DATA_BLOCK "n0008-icg12-el001-k30001_SN51_3"   // DB1076, F_DB
VERSION : 0.1
// stored: AutoNumber true, DBAccessibleFromOPCUA true, DBAccessibleFromWebserver true, InstanceOfName 00_Push-Button_Input, InstanceOfType FB
"00_Push-Button_Input"
   // VAR_INPUT
   //    IN_1 : Bool;
   //    IN_2 : Bool;
   //    IN_3 : Bool;
   //    IN_4 : Bool;
   //    ON_Tristate : Bool;
   //    ON_Lamp : Bool;
   //    Reset : Bool;
   //    REAC_DELAY { ExternalWritable := 'False'} : Time;
   //    Bypass_ET200 : Bool;
   // END_VAR
   // VAR_OUTPUT
   //    OUT_1 : Bool;
   //    OUT_2 : Bool;
   //    OUT_3 : Bool;
   //    OUT_4 : Bool;
   //    Diag_1 : Bool;
   //    Diag_2 : Bool;
   //    Diag_3 : Bool;
   //    Diag_4 : Bool;
   //    Lamp_1 : Bool;
   //    Lamp_2 : Bool;
   //    Lamp_3 : Bool;
   //    Lamp_4 : Bool;
   // END_VAR
   // VAR
   //    ESTOP_1 { S7_SetPoint := 'True'} : ESTOP1;
   //    ESTOP_2 { S7_SetPoint := 'True'} : ESTOP1;
   //    ESTOP_3 { S7_SetPoint := 'True'} : ESTOP1;
   //    ESTOP_4 { S7_SetPoint := 'True'} : ESTOP1;
   //    TON_1 { ExternalWritable := 'False'} : TON;
   //    TON_2 { ExternalWritable := 'False'} : TON;
   //    TON_3 { ExternalWritable := 'False'} : TON;
   //    TON_4 { ExternalWritable := 'False'} : TON;
   // END_VAR
BEGIN
END_DATA_BLOCK

DATA_BLOCK "n0008-icg12-el001-k30001_SN51_4"   // DB1077, F_DB
VERSION : 0.1
// stored: AutoNumber true, DBAccessibleFromOPCUA true, DBAccessibleFromWebserver true, InstanceOfName 00_Push-Button_Input, InstanceOfType FB
"00_Push-Button_Input"
   // VAR_INPUT
   //    IN_1 : Bool;
   //    IN_2 : Bool;
   //    IN_3 : Bool;
   //    IN_4 : Bool;
   //    ON_Tristate : Bool;
   //    ON_Lamp : Bool;
   //    Reset : Bool;
   //    REAC_DELAY { ExternalWritable := 'False'} : Time;
   //    Bypass_ET200 : Bool;
   // END_VAR
   // VAR_OUTPUT
   //    OUT_1 : Bool;
   //    OUT_2 : Bool;
   //    OUT_3 : Bool;
   //    OUT_4 : Bool;
   //    Diag_1 : Bool;
   //    Diag_2 : Bool;
   //    Diag_3 : Bool;
   //    Diag_4 : Bool;
   //    Lamp_1 : Bool;
   //    Lamp_2 : Bool;
   //    Lamp_3 : Bool;
   //    Lamp_4 : Bool;
   // END_VAR
   // VAR
   //    ESTOP_1 { S7_SetPoint := 'True'} : ESTOP1;
   //    ESTOP_2 { S7_SetPoint := 'True'} : ESTOP1;
   //    ESTOP_3 { S7_SetPoint := 'True'} : ESTOP1;
   //    ESTOP_4 { S7_SetPoint := 'True'} : ESTOP1;
   //    TON_1 { ExternalWritable := 'False'} : TON;
   //    TON_2 { ExternalWritable := 'False'} : TON;
   //    TON_3 { ExternalWritable := 'False'} : TON;
   //    TON_4 { ExternalWritable := 'False'} : TON;
   // END_VAR
BEGIN
END_DATA_BLOCK

DATA_BLOCK "n0026-uc915-xn10_SN51_1"   // DB1078, F_DB
VERSION : 0.1
// stored: AutoNumber true, DBAccessibleFromOPCUA true, DBAccessibleFromWebserver true, InstanceOfName 00_Push-Button_Input, InstanceOfType FB
"00_Push-Button_Input"
   // VAR_INPUT
   //    IN_1 : Bool;
   //    IN_2 : Bool;
   //    IN_3 : Bool;
   //    IN_4 : Bool;
   //    ON_Tristate : Bool;
   //    ON_Lamp : Bool;
   //    Reset : Bool;
   //    REAC_DELAY { ExternalWritable := 'False'} : Time;
   //    Bypass_ET200 : Bool;
   // END_VAR
   // VAR_OUTPUT
   //    OUT_1 : Bool;
   //    OUT_2 : Bool;
   //    OUT_3 : Bool;
   //    OUT_4 : Bool;
   //    Diag_1 : Bool;
   //    Diag_2 : Bool;
   //    Diag_3 : Bool;
   //    Diag_4 : Bool;
   //    Lamp_1 : Bool;
   //    Lamp_2 : Bool;
   //    Lamp_3 : Bool;
   //    Lamp_4 : Bool;
   // END_VAR
   // VAR
   //    ESTOP_1 { S7_SetPoint := 'True'} : ESTOP1;
   //    ESTOP_2 { S7_SetPoint := 'True'} : ESTOP1;
   //    ESTOP_3 { S7_SetPoint := 'True'} : ESTOP1;
   //    ESTOP_4 { S7_SetPoint := 'True'} : ESTOP1;
   //    TON_1 { ExternalWritable := 'False'} : TON;
   //    TON_2 { ExternalWritable := 'False'} : TON;
   //    TON_3 { ExternalWritable := 'False'} : TON;
   //    TON_4 { ExternalWritable := 'False'} : TON;
   // END_VAR
BEGIN
END_DATA_BLOCK

DATA_BLOCK "n0026-uc915-xn10_SN51_2"   // DB1079, F_DB
VERSION : 0.1
// stored: AutoNumber true, DBAccessibleFromOPCUA true, DBAccessibleFromWebserver true, InstanceOfName 00_Push-Button_Input, InstanceOfType FB
"00_Push-Button_Input"
   // VAR_INPUT
   //    IN_1 : Bool;
   //    IN_2 : Bool;
   //    IN_3 : Bool;
   //    IN_4 : Bool;
   //    ON_Tristate : Bool;
   //    ON_Lamp : Bool;
   //    Reset : Bool;
   //    REAC_DELAY { ExternalWritable := 'False'} : Time;
   //    Bypass_ET200 : Bool;
   // END_VAR
   // VAR_OUTPUT
   //    OUT_1 : Bool;
   //    OUT_2 : Bool;
   //    OUT_3 : Bool;
   //    OUT_4 : Bool;
   //    Diag_1 : Bool;
   //    Diag_2 : Bool;
   //    Diag_3 : Bool;
   //    Diag_4 : Bool;
   //    Lamp_1 : Bool;
   //    Lamp_2 : Bool;
   //    Lamp_3 : Bool;
   //    Lamp_4 : Bool;
   // END_VAR
   // VAR
   //    ESTOP_1 { S7_SetPoint := 'True'} : ESTOP1;
   //    ESTOP_2 { S7_SetPoint := 'True'} : ESTOP1;
   //    ESTOP_3 { S7_SetPoint := 'True'} : ESTOP1;
   //    ESTOP_4 { S7_SetPoint := 'True'} : ESTOP1;
   //    TON_1 { ExternalWritable := 'False'} : TON;
   //    TON_2 { ExternalWritable := 'False'} : TON;
   //    TON_3 { ExternalWritable := 'False'} : TON;
   //    TON_4 { ExternalWritable := 'False'} : TON;
   // END_VAR
BEGIN
END_DATA_BLOCK

DATA_BLOCK "n0027-uc915-xn11_SN51_1"   // DB1080, F_DB
VERSION : 0.1
// stored: AutoNumber true, DBAccessibleFromOPCUA true, DBAccessibleFromWebserver true, InstanceOfName 00_Push-Button_Input, InstanceOfType FB
"00_Push-Button_Input"
   // VAR_INPUT
   //    IN_1 : Bool;
   //    IN_2 : Bool;
   //    IN_3 : Bool;
   //    IN_4 : Bool;
   //    ON_Tristate : Bool;
   //    ON_Lamp : Bool;
   //    Reset : Bool;
   //    REAC_DELAY { ExternalWritable := 'False'} : Time;
   //    Bypass_ET200 : Bool;
   // END_VAR
   // VAR_OUTPUT
   //    OUT_1 : Bool;
   //    OUT_2 : Bool;
   //    OUT_3 : Bool;
   //    OUT_4 : Bool;
   //    Diag_1 : Bool;
   //    Diag_2 : Bool;
   //    Diag_3 : Bool;
   //    Diag_4 : Bool;
   //    Lamp_1 : Bool;
   //    Lamp_2 : Bool;
   //    Lamp_3 : Bool;
   //    Lamp_4 : Bool;
   // END_VAR
   // VAR
   //    ESTOP_1 { S7_SetPoint := 'True'} : ESTOP1;
   //    ESTOP_2 { S7_SetPoint := 'True'} : ESTOP1;
   //    ESTOP_3 { S7_SetPoint := 'True'} : ESTOP1;
   //    ESTOP_4 { S7_SetPoint := 'True'} : ESTOP1;
   //    TON_1 { ExternalWritable := 'False'} : TON;
   //    TON_2 { ExternalWritable := 'False'} : TON;
   //    TON_3 { ExternalWritable := 'False'} : TON;
   //    TON_4 { ExternalWritable := 'False'} : TON;
   // END_VAR
BEGIN
END_DATA_BLOCK

DATA_BLOCK "n0029-ct2-el001-k30001_SN51_1"   // DB1081, F_DB
VERSION : 0.1
// stored: AutoNumber true, DBAccessibleFromOPCUA true, DBAccessibleFromWebserver true, InstanceOfName 00_Push-Button_Input, InstanceOfType FB
"00_Push-Button_Input"
   // VAR_INPUT
   //    IN_1 : Bool;
   //    IN_2 : Bool;
   //    IN_3 : Bool;
   //    IN_4 : Bool;
   //    ON_Tristate : Bool;
   //    ON_Lamp : Bool;
   //    Reset : Bool;
   //    REAC_DELAY { ExternalWritable := 'False'} : Time;
   //    Bypass_ET200 : Bool;
   // END_VAR
   // VAR_OUTPUT
   //    OUT_1 : Bool;
   //    OUT_2 : Bool;
   //    OUT_3 : Bool;
   //    OUT_4 : Bool;
   //    Diag_1 : Bool;
   //    Diag_2 : Bool;
   //    Diag_3 : Bool;
   //    Diag_4 : Bool;
   //    Lamp_1 : Bool;
   //    Lamp_2 : Bool;
   //    Lamp_3 : Bool;
   //    Lamp_4 : Bool;
   // END_VAR
   // VAR
   //    ESTOP_1 { S7_SetPoint := 'True'} : ESTOP1;
   //    ESTOP_2 { S7_SetPoint := 'True'} : ESTOP1;
   //    ESTOP_3 { S7_SetPoint := 'True'} : ESTOP1;
   //    ESTOP_4 { S7_SetPoint := 'True'} : ESTOP1;
   //    TON_1 { ExternalWritable := 'False'} : TON;
   //    TON_2 { ExternalWritable := 'False'} : TON;
   //    TON_3 { ExternalWritable := 'False'} : TON;
   //    TON_4 { ExternalWritable := 'False'} : TON;
   // END_VAR
BEGIN
END_DATA_BLOCK

DATA_BLOCK "n0029-ct2-el001-k30001_SN51_2"   // DB1082, F_DB
VERSION : 0.1
// stored: AutoNumber true, DBAccessibleFromOPCUA true, DBAccessibleFromWebserver true, InstanceOfName 00_Push-Button_Input, InstanceOfType FB
"00_Push-Button_Input"
   // VAR_INPUT
   //    IN_1 : Bool;
   //    IN_2 : Bool;
   //    IN_3 : Bool;
   //    IN_4 : Bool;
   //    ON_Tristate : Bool;
   //    ON_Lamp : Bool;
   //    Reset : Bool;
   //    REAC_DELAY { ExternalWritable := 'False'} : Time;
   //    Bypass_ET200 : Bool;
   // END_VAR
   // VAR_OUTPUT
   //    OUT_1 : Bool;
   //    OUT_2 : Bool;
   //    OUT_3 : Bool;
   //    OUT_4 : Bool;
   //    Diag_1 : Bool;
   //    Diag_2 : Bool;
   //    Diag_3 : Bool;
   //    Diag_4 : Bool;
   //    Lamp_1 : Bool;
   //    Lamp_2 : Bool;
   //    Lamp_3 : Bool;
   //    Lamp_4 : Bool;
   // END_VAR
   // VAR
   //    ESTOP_1 { S7_SetPoint := 'True'} : ESTOP1;
   //    ESTOP_2 { S7_SetPoint := 'True'} : ESTOP1;
   //    ESTOP_3 { S7_SetPoint := 'True'} : ESTOP1;
   //    ESTOP_4 { S7_SetPoint := 'True'} : ESTOP1;
   //    TON_1 { ExternalWritable := 'False'} : TON;
   //    TON_2 { ExternalWritable := 'False'} : TON;
   //    TON_3 { ExternalWritable := 'False'} : TON;
   //    TON_4 { ExternalWritable := 'False'} : TON;
   // END_VAR
BEGIN
END_DATA_BLOCK

DATA_BLOCK "n0029-ct2-el001-k30001_SN51_3"   // DB1083, F_DB
VERSION : 0.1
// stored: AutoNumber true, DBAccessibleFromOPCUA true, DBAccessibleFromWebserver true, InstanceOfName 00_Push-Button_Input, InstanceOfType FB
"00_Push-Button_Input"
   // VAR_INPUT
   //    IN_1 : Bool;
   //    IN_2 : Bool;
   //    IN_3 : Bool;
   //    IN_4 : Bool;
   //    ON_Tristate : Bool;
   //    ON_Lamp : Bool;
   //    Reset : Bool;
   //    REAC_DELAY { ExternalWritable := 'False'} : Time;
   //    Bypass_ET200 : Bool;
   // END_VAR
   // VAR_OUTPUT
   //    OUT_1 : Bool;
   //    OUT_2 : Bool;
   //    OUT_3 : Bool;
   //    OUT_4 : Bool;
   //    Diag_1 : Bool;
   //    Diag_2 : Bool;
   //    Diag_3 : Bool;
   //    Diag_4 : Bool;
   //    Lamp_1 : Bool;
   //    Lamp_2 : Bool;
   //    Lamp_3 : Bool;
   //    Lamp_4 : Bool;
   // END_VAR
   // VAR
   //    ESTOP_1 { S7_SetPoint := 'True'} : ESTOP1;
   //    ESTOP_2 { S7_SetPoint := 'True'} : ESTOP1;
   //    ESTOP_3 { S7_SetPoint := 'True'} : ESTOP1;
   //    ESTOP_4 { S7_SetPoint := 'True'} : ESTOP1;
   //    TON_1 { ExternalWritable := 'False'} : TON;
   //    TON_2 { ExternalWritable := 'False'} : TON;
   //    TON_3 { ExternalWritable := 'False'} : TON;
   //    TON_4 { ExternalWritable := 'False'} : TON;
   // END_VAR
BEGIN
END_DATA_BLOCK

DATA_BLOCK "n0029-ct2-el001-k30001_SN51_4"   // DB1084, F_DB
VERSION : 0.1
// stored: AutoNumber true, DBAccessibleFromOPCUA true, DBAccessibleFromWebserver true, InstanceOfName 00_Push-Button_Input, InstanceOfType FB
"00_Push-Button_Input"
   // VAR_INPUT
   //    IN_1 : Bool;
   //    IN_2 : Bool;
   //    IN_3 : Bool;
   //    IN_4 : Bool;
   //    ON_Tristate : Bool;
   //    ON_Lamp : Bool;
   //    Reset : Bool;
   //    REAC_DELAY { ExternalWritable := 'False'} : Time;
   //    Bypass_ET200 : Bool;
   // END_VAR
   // VAR_OUTPUT
   //    OUT_1 : Bool;
   //    OUT_2 : Bool;
   //    OUT_3 : Bool;
   //    OUT_4 : Bool;
   //    Diag_1 : Bool;
   //    Diag_2 : Bool;
   //    Diag_3 : Bool;
   //    Diag_4 : Bool;
   //    Lamp_1 : Bool;
   //    Lamp_2 : Bool;
   //    Lamp_3 : Bool;
   //    Lamp_4 : Bool;
   // END_VAR
   // VAR
   //    ESTOP_1 { S7_SetPoint := 'True'} : ESTOP1;
   //    ESTOP_2 { S7_SetPoint := 'True'} : ESTOP1;
   //    ESTOP_3 { S7_SetPoint := 'True'} : ESTOP1;
   //    ESTOP_4 { S7_SetPoint := 'True'} : ESTOP1;
   //    TON_1 { ExternalWritable := 'False'} : TON;
   //    TON_2 { ExternalWritable := 'False'} : TON;
   //    TON_3 { ExternalWritable := 'False'} : TON;
   //    TON_4 { ExternalWritable := 'False'} : TON;
   // END_VAR
BEGIN
END_DATA_BLOCK

DATA_BLOCK "n0029-ct2-el001-k30001_SN51_5"   // DB1085, F_DB
VERSION : 0.1
// stored: AutoNumber true, DBAccessibleFromOPCUA true, DBAccessibleFromWebserver true, InstanceOfName 00_Push-Button_Input, InstanceOfType FB
"00_Push-Button_Input"
   // VAR_INPUT
   //    IN_1 : Bool;
   //    IN_2 : Bool;
   //    IN_3 : Bool;
   //    IN_4 : Bool;
   //    ON_Tristate : Bool;
   //    ON_Lamp : Bool;
   //    Reset : Bool;
   //    REAC_DELAY { ExternalWritable := 'False'} : Time;
   //    Bypass_ET200 : Bool;
   // END_VAR
   // VAR_OUTPUT
   //    OUT_1 : Bool;
   //    OUT_2 : Bool;
   //    OUT_3 : Bool;
   //    OUT_4 : Bool;
   //    Diag_1 : Bool;
   //    Diag_2 : Bool;
   //    Diag_3 : Bool;
   //    Diag_4 : Bool;
   //    Lamp_1 : Bool;
   //    Lamp_2 : Bool;
   //    Lamp_3 : Bool;
   //    Lamp_4 : Bool;
   // END_VAR
   // VAR
   //    ESTOP_1 { S7_SetPoint := 'True'} : ESTOP1;
   //    ESTOP_2 { S7_SetPoint := 'True'} : ESTOP1;
   //    ESTOP_3 { S7_SetPoint := 'True'} : ESTOP1;
   //    ESTOP_4 { S7_SetPoint := 'True'} : ESTOP1;
   //    TON_1 { ExternalWritable := 'False'} : TON;
   //    TON_2 { ExternalWritable := 'False'} : TON;
   //    TON_3 { ExternalWritable := 'False'} : TON;
   //    TON_4 { ExternalWritable := 'False'} : TON;
   // END_VAR
BEGIN
END_DATA_BLOCK

DATA_BLOCK "n0033-uc26-el001-k30001_SN51_1"   // DB1086, F_DB
VERSION : 0.1
// stored: AutoNumber true, DBAccessibleFromOPCUA true, DBAccessibleFromWebserver true, InstanceOfName 00_Push-Button_Input, InstanceOfType FB
"00_Push-Button_Input"
   // VAR_INPUT
   //    IN_1 : Bool;
   //    IN_2 : Bool;
   //    IN_3 : Bool;
   //    IN_4 : Bool;
   //    ON_Tristate : Bool;
   //    ON_Lamp : Bool;
   //    Reset : Bool;
   //    REAC_DELAY { ExternalWritable := 'False'} : Time;
   //    Bypass_ET200 : Bool;
   // END_VAR
   // VAR_OUTPUT
   //    OUT_1 : Bool;
   //    OUT_2 : Bool;
   //    OUT_3 : Bool;
   //    OUT_4 : Bool;
   //    Diag_1 : Bool;
   //    Diag_2 : Bool;
   //    Diag_3 : Bool;
   //    Diag_4 : Bool;
   //    Lamp_1 : Bool;
   //    Lamp_2 : Bool;
   //    Lamp_3 : Bool;
   //    Lamp_4 : Bool;
   // END_VAR
   // VAR
   //    ESTOP_1 { S7_SetPoint := 'True'} : ESTOP1;
   //    ESTOP_2 { S7_SetPoint := 'True'} : ESTOP1;
   //    ESTOP_3 { S7_SetPoint := 'True'} : ESTOP1;
   //    ESTOP_4 { S7_SetPoint := 'True'} : ESTOP1;
   //    TON_1 { ExternalWritable := 'False'} : TON;
   //    TON_2 { ExternalWritable := 'False'} : TON;
   //    TON_3 { ExternalWritable := 'False'} : TON;
   //    TON_4 { ExternalWritable := 'False'} : TON;
   // END_VAR
BEGIN
END_DATA_BLOCK

DATA_BLOCK "n0033-uc26-el001-k30001_SN51_2"   // DB1087, F_DB
VERSION : 0.1
// stored: AutoNumber true, DBAccessibleFromOPCUA true, DBAccessibleFromWebserver true, InstanceOfName 00_Push-Button_Input, InstanceOfType FB
"00_Push-Button_Input"
   // VAR_INPUT
   //    IN_1 : Bool;
   //    IN_2 : Bool;
   //    IN_3 : Bool;
   //    IN_4 : Bool;
   //    ON_Tristate : Bool;
   //    ON_Lamp : Bool;
   //    Reset : Bool;
   //    REAC_DELAY { ExternalWritable := 'False'} : Time;
   //    Bypass_ET200 : Bool;
   // END_VAR
   // VAR_OUTPUT
   //    OUT_1 : Bool;
   //    OUT_2 : Bool;
   //    OUT_3 : Bool;
   //    OUT_4 : Bool;
   //    Diag_1 : Bool;
   //    Diag_2 : Bool;
   //    Diag_3 : Bool;
   //    Diag_4 : Bool;
   //    Lamp_1 : Bool;
   //    Lamp_2 : Bool;
   //    Lamp_3 : Bool;
   //    Lamp_4 : Bool;
   // END_VAR
   // VAR
   //    ESTOP_1 { S7_SetPoint := 'True'} : ESTOP1;
   //    ESTOP_2 { S7_SetPoint := 'True'} : ESTOP1;
   //    ESTOP_3 { S7_SetPoint := 'True'} : ESTOP1;
   //    ESTOP_4 { S7_SetPoint := 'True'} : ESTOP1;
   //    TON_1 { ExternalWritable := 'False'} : TON;
   //    TON_2 { ExternalWritable := 'False'} : TON;
   //    TON_3 { ExternalWritable := 'False'} : TON;
   //    TON_4 { ExternalWritable := 'False'} : TON;
   // END_VAR
BEGIN
END_DATA_BLOCK

DATA_BLOCK "n0033-uc26-el001-k30001_SN51_3"   // DB1088, F_DB
VERSION : 0.1
// stored: AutoNumber true, DBAccessibleFromOPCUA true, DBAccessibleFromWebserver true, InstanceOfName 00_Push-Button_Input, InstanceOfType FB
"00_Push-Button_Input"
   // VAR_INPUT
   //    IN_1 : Bool;
   //    IN_2 : Bool;
   //    IN_3 : Bool;
   //    IN_4 : Bool;
   //    ON_Tristate : Bool;
   //    ON_Lamp : Bool;
   //    Reset : Bool;
   //    REAC_DELAY { ExternalWritable := 'False'} : Time;
   //    Bypass_ET200 : Bool;
   // END_VAR
   // VAR_OUTPUT
   //    OUT_1 : Bool;
   //    OUT_2 : Bool;
   //    OUT_3 : Bool;
   //    OUT_4 : Bool;
   //    Diag_1 : Bool;
   //    Diag_2 : Bool;
   //    Diag_3 : Bool;
   //    Diag_4 : Bool;
   //    Lamp_1 : Bool;
   //    Lamp_2 : Bool;
   //    Lamp_3 : Bool;
   //    Lamp_4 : Bool;
   // END_VAR
   // VAR
   //    ESTOP_1 { S7_SetPoint := 'True'} : ESTOP1;
   //    ESTOP_2 { S7_SetPoint := 'True'} : ESTOP1;
   //    ESTOP_3 { S7_SetPoint := 'True'} : ESTOP1;
   //    ESTOP_4 { S7_SetPoint := 'True'} : ESTOP1;
   //    TON_1 { ExternalWritable := 'False'} : TON;
   //    TON_2 { ExternalWritable := 'False'} : TON;
   //    TON_3 { ExternalWritable := 'False'} : TON;
   //    TON_4 { ExternalWritable := 'False'} : TON;
   // END_VAR
BEGIN
END_DATA_BLOCK

DATA_BLOCK "n0034-uc264-xn10_SN51_1"   // DB1089, F_DB
VERSION : 0.1
// stored: AutoNumber true, DBAccessibleFromOPCUA true, DBAccessibleFromWebserver true, InstanceOfName 00_Push-Button_Input, InstanceOfType FB
"00_Push-Button_Input"
   // VAR_INPUT
   //    IN_1 : Bool;
   //    IN_2 : Bool;
   //    IN_3 : Bool;
   //    IN_4 : Bool;
   //    ON_Tristate : Bool;
   //    ON_Lamp : Bool;
   //    Reset : Bool;
   //    REAC_DELAY { ExternalWritable := 'False'} : Time;
   //    Bypass_ET200 : Bool;
   // END_VAR
   // VAR_OUTPUT
   //    OUT_1 : Bool;
   //    OUT_2 : Bool;
   //    OUT_3 : Bool;
   //    OUT_4 : Bool;
   //    Diag_1 : Bool;
   //    Diag_2 : Bool;
   //    Diag_3 : Bool;
   //    Diag_4 : Bool;
   //    Lamp_1 : Bool;
   //    Lamp_2 : Bool;
   //    Lamp_3 : Bool;
   //    Lamp_4 : Bool;
   // END_VAR
   // VAR
   //    ESTOP_1 { S7_SetPoint := 'True'} : ESTOP1;
   //    ESTOP_2 { S7_SetPoint := 'True'} : ESTOP1;
   //    ESTOP_3 { S7_SetPoint := 'True'} : ESTOP1;
   //    ESTOP_4 { S7_SetPoint := 'True'} : ESTOP1;
   //    TON_1 { ExternalWritable := 'False'} : TON;
   //    TON_2 { ExternalWritable := 'False'} : TON;
   //    TON_3 { ExternalWritable := 'False'} : TON;
   //    TON_4 { ExternalWritable := 'False'} : TON;
   // END_VAR
BEGIN
END_DATA_BLOCK

DATA_BLOCK "n0034-uc264-xn10_SN51_2"   // DB1090, F_DB
VERSION : 0.1
// stored: AutoNumber true, DBAccessibleFromOPCUA true, DBAccessibleFromWebserver true, InstanceOfName 00_Push-Button_Input, InstanceOfType FB
"00_Push-Button_Input"
   // VAR_INPUT
   //    IN_1 : Bool;
   //    IN_2 : Bool;
   //    IN_3 : Bool;
   //    IN_4 : Bool;
   //    ON_Tristate : Bool;
   //    ON_Lamp : Bool;
   //    Reset : Bool;
   //    REAC_DELAY { ExternalWritable := 'False'} : Time;
   //    Bypass_ET200 : Bool;
   // END_VAR
   // VAR_OUTPUT
   //    OUT_1 : Bool;
   //    OUT_2 : Bool;
   //    OUT_3 : Bool;
   //    OUT_4 : Bool;
   //    Diag_1 : Bool;
   //    Diag_2 : Bool;
   //    Diag_3 : Bool;
   //    Diag_4 : Bool;
   //    Lamp_1 : Bool;
   //    Lamp_2 : Bool;
   //    Lamp_3 : Bool;
   //    Lamp_4 : Bool;
   // END_VAR
   // VAR
   //    ESTOP_1 { S7_SetPoint := 'True'} : ESTOP1;
   //    ESTOP_2 { S7_SetPoint := 'True'} : ESTOP1;
   //    ESTOP_3 { S7_SetPoint := 'True'} : ESTOP1;
   //    ESTOP_4 { S7_SetPoint := 'True'} : ESTOP1;
   //    TON_1 { ExternalWritable := 'False'} : TON;
   //    TON_2 { ExternalWritable := 'False'} : TON;
   //    TON_3 { ExternalWritable := 'False'} : TON;
   //    TON_4 { ExternalWritable := 'False'} : TON;
   // END_VAR
BEGIN
END_DATA_BLOCK

DATA_BLOCK "n0035-ct2-el002-k30001_SN51_1"   // DB1091, F_DB
VERSION : 0.1
// stored: AutoNumber true, DBAccessibleFromOPCUA true, DBAccessibleFromWebserver true, InstanceOfName 00_Push-Button_Input, InstanceOfType FB
"00_Push-Button_Input"
   // VAR_INPUT
   //    IN_1 : Bool;
   //    IN_2 : Bool;
   //    IN_3 : Bool;
   //    IN_4 : Bool;
   //    ON_Tristate : Bool;
   //    ON_Lamp : Bool;
   //    Reset : Bool;
   //    REAC_DELAY { ExternalWritable := 'False'} : Time;
   //    Bypass_ET200 : Bool;
   // END_VAR
   // VAR_OUTPUT
   //    OUT_1 : Bool;
   //    OUT_2 : Bool;
   //    OUT_3 : Bool;
   //    OUT_4 : Bool;
   //    Diag_1 : Bool;
   //    Diag_2 : Bool;
   //    Diag_3 : Bool;
   //    Diag_4 : Bool;
   //    Lamp_1 : Bool;
   //    Lamp_2 : Bool;
   //    Lamp_3 : Bool;
   //    Lamp_4 : Bool;
   // END_VAR
   // VAR
   //    ESTOP_1 { S7_SetPoint := 'True'} : ESTOP1;
   //    ESTOP_2 { S7_SetPoint := 'True'} : ESTOP1;
   //    ESTOP_3 { S7_SetPoint := 'True'} : ESTOP1;
   //    ESTOP_4 { S7_SetPoint := 'True'} : ESTOP1;
   //    TON_1 { ExternalWritable := 'False'} : TON;
   //    TON_2 { ExternalWritable := 'False'} : TON;
   //    TON_3 { ExternalWritable := 'False'} : TON;
   //    TON_4 { ExternalWritable := 'False'} : TON;
   // END_VAR
BEGIN
END_DATA_BLOCK

DATA_BLOCK "n0035-ct2-el002-k30001_SN51_2"   // DB1092, F_DB
VERSION : 0.1
// stored: AutoNumber true, DBAccessibleFromOPCUA true, DBAccessibleFromWebserver true, InstanceOfName 00_Push-Button_Input, InstanceOfType FB
"00_Push-Button_Input"
   // VAR_INPUT
   //    IN_1 : Bool;
   //    IN_2 : Bool;
   //    IN_3 : Bool;
   //    IN_4 : Bool;
   //    ON_Tristate : Bool;
   //    ON_Lamp : Bool;
   //    Reset : Bool;
   //    REAC_DELAY { ExternalWritable := 'False'} : Time;
   //    Bypass_ET200 : Bool;
   // END_VAR
   // VAR_OUTPUT
   //    OUT_1 : Bool;
   //    OUT_2 : Bool;
   //    OUT_3 : Bool;
   //    OUT_4 : Bool;
   //    Diag_1 : Bool;
   //    Diag_2 : Bool;
   //    Diag_3 : Bool;
   //    Diag_4 : Bool;
   //    Lamp_1 : Bool;
   //    Lamp_2 : Bool;
   //    Lamp_3 : Bool;
   //    Lamp_4 : Bool;
   // END_VAR
   // VAR
   //    ESTOP_1 { S7_SetPoint := 'True'} : ESTOP1;
   //    ESTOP_2 { S7_SetPoint := 'True'} : ESTOP1;
   //    ESTOP_3 { S7_SetPoint := 'True'} : ESTOP1;
   //    ESTOP_4 { S7_SetPoint := 'True'} : ESTOP1;
   //    TON_1 { ExternalWritable := 'False'} : TON;
   //    TON_2 { ExternalWritable := 'False'} : TON;
   //    TON_3 { ExternalWritable := 'False'} : TON;
   //    TON_4 { ExternalWritable := 'False'} : TON;
   // END_VAR
BEGIN
END_DATA_BLOCK

DATA_BLOCK "n0035-ct2-el002-k30001_SN51_3"   // DB1093, F_DB
VERSION : 0.1
// stored: AutoNumber true, DBAccessibleFromOPCUA true, DBAccessibleFromWebserver true, InstanceOfName 00_Push-Button_Input, InstanceOfType FB
"00_Push-Button_Input"
   // VAR_INPUT
   //    IN_1 : Bool;
   //    IN_2 : Bool;
   //    IN_3 : Bool;
   //    IN_4 : Bool;
   //    ON_Tristate : Bool;
   //    ON_Lamp : Bool;
   //    Reset : Bool;
   //    REAC_DELAY { ExternalWritable := 'False'} : Time;
   //    Bypass_ET200 : Bool;
   // END_VAR
   // VAR_OUTPUT
   //    OUT_1 : Bool;
   //    OUT_2 : Bool;
   //    OUT_3 : Bool;
   //    OUT_4 : Bool;
   //    Diag_1 : Bool;
   //    Diag_2 : Bool;
   //    Diag_3 : Bool;
   //    Diag_4 : Bool;
   //    Lamp_1 : Bool;
   //    Lamp_2 : Bool;
   //    Lamp_3 : Bool;
   //    Lamp_4 : Bool;
   // END_VAR
   // VAR
   //    ESTOP_1 { S7_SetPoint := 'True'} : ESTOP1;
   //    ESTOP_2 { S7_SetPoint := 'True'} : ESTOP1;
   //    ESTOP_3 { S7_SetPoint := 'True'} : ESTOP1;
   //    ESTOP_4 { S7_SetPoint := 'True'} : ESTOP1;
   //    TON_1 { ExternalWritable := 'False'} : TON;
   //    TON_2 { ExternalWritable := 'False'} : TON;
   //    TON_3 { ExternalWritable := 'False'} : TON;
   //    TON_4 { ExternalWritable := 'False'} : TON;
   // END_VAR
BEGIN
END_DATA_BLOCK

DATA_BLOCK "n0035-ct2-el002-k30001_SN51_4"   // DB1094, F_DB
VERSION : 0.1
// stored: AutoNumber true, DBAccessibleFromOPCUA true, DBAccessibleFromWebserver true, InstanceOfName 00_Push-Button_Input, InstanceOfType FB
"00_Push-Button_Input"
   // VAR_INPUT
   //    IN_1 : Bool;
   //    IN_2 : Bool;
   //    IN_3 : Bool;
   //    IN_4 : Bool;
   //    ON_Tristate : Bool;
   //    ON_Lamp : Bool;
   //    Reset : Bool;
   //    REAC_DELAY { ExternalWritable := 'False'} : Time;
   //    Bypass_ET200 : Bool;
   // END_VAR
   // VAR_OUTPUT
   //    OUT_1 : Bool;
   //    OUT_2 : Bool;
   //    OUT_3 : Bool;
   //    OUT_4 : Bool;
   //    Diag_1 : Bool;
   //    Diag_2 : Bool;
   //    Diag_3 : Bool;
   //    Diag_4 : Bool;
   //    Lamp_1 : Bool;
   //    Lamp_2 : Bool;
   //    Lamp_3 : Bool;
   //    Lamp_4 : Bool;
   // END_VAR
   // VAR
   //    ESTOP_1 { S7_SetPoint := 'True'} : ESTOP1;
   //    ESTOP_2 { S7_SetPoint := 'True'} : ESTOP1;
   //    ESTOP_3 { S7_SetPoint := 'True'} : ESTOP1;
   //    ESTOP_4 { S7_SetPoint := 'True'} : ESTOP1;
   //    TON_1 { ExternalWritable := 'False'} : TON;
   //    TON_2 { ExternalWritable := 'False'} : TON;
   //    TON_3 { ExternalWritable := 'False'} : TON;
   //    TON_4 { ExternalWritable := 'False'} : TON;
   // END_VAR
BEGIN
END_DATA_BLOCK

DATA_BLOCK "n0035-ct2-el002-k30001_SN51_5"   // DB1095, F_DB
VERSION : 0.1
// stored: AutoNumber true, DBAccessibleFromOPCUA true, DBAccessibleFromWebserver true, InstanceOfName 00_Push-Button_Input, InstanceOfType FB
"00_Push-Button_Input"
   // VAR_INPUT
   //    IN_1 : Bool;
   //    IN_2 : Bool;
   //    IN_3 : Bool;
   //    IN_4 : Bool;
   //    ON_Tristate : Bool;
   //    ON_Lamp : Bool;
   //    Reset : Bool;
   //    REAC_DELAY { ExternalWritable := 'False'} : Time;
   //    Bypass_ET200 : Bool;
   // END_VAR
   // VAR_OUTPUT
   //    OUT_1 : Bool;
   //    OUT_2 : Bool;
   //    OUT_3 : Bool;
   //    OUT_4 : Bool;
   //    Diag_1 : Bool;
   //    Diag_2 : Bool;
   //    Diag_3 : Bool;
   //    Diag_4 : Bool;
   //    Lamp_1 : Bool;
   //    Lamp_2 : Bool;
   //    Lamp_3 : Bool;
   //    Lamp_4 : Bool;
   // END_VAR
   // VAR
   //    ESTOP_1 { S7_SetPoint := 'True'} : ESTOP1;
   //    ESTOP_2 { S7_SetPoint := 'True'} : ESTOP1;
   //    ESTOP_3 { S7_SetPoint := 'True'} : ESTOP1;
   //    ESTOP_4 { S7_SetPoint := 'True'} : ESTOP1;
   //    TON_1 { ExternalWritable := 'False'} : TON;
   //    TON_2 { ExternalWritable := 'False'} : TON;
   //    TON_3 { ExternalWritable := 'False'} : TON;
   //    TON_4 { ExternalWritable := 'False'} : TON;
   // END_VAR
BEGIN
END_DATA_BLOCK

DATA_BLOCK "n0041-uc27-el001-k30001_SN51_1"   // DB1096, F_DB
VERSION : 0.1
// stored: AutoNumber true, DBAccessibleFromOPCUA true, DBAccessibleFromWebserver true, InstanceOfName 00_Push-Button_Input, InstanceOfType FB
"00_Push-Button_Input"
   // VAR_INPUT
   //    IN_1 : Bool;
   //    IN_2 : Bool;
   //    IN_3 : Bool;
   //    IN_4 : Bool;
   //    ON_Tristate : Bool;
   //    ON_Lamp : Bool;
   //    Reset : Bool;
   //    REAC_DELAY { ExternalWritable := 'False'} : Time;
   //    Bypass_ET200 : Bool;
   // END_VAR
   // VAR_OUTPUT
   //    OUT_1 : Bool;
   //    OUT_2 : Bool;
   //    OUT_3 : Bool;
   //    OUT_4 : Bool;
   //    Diag_1 : Bool;
   //    Diag_2 : Bool;
   //    Diag_3 : Bool;
   //    Diag_4 : Bool;
   //    Lamp_1 : Bool;
   //    Lamp_2 : Bool;
   //    Lamp_3 : Bool;
   //    Lamp_4 : Bool;
   // END_VAR
   // VAR
   //    ESTOP_1 { S7_SetPoint := 'True'} : ESTOP1;
   //    ESTOP_2 { S7_SetPoint := 'True'} : ESTOP1;
   //    ESTOP_3 { S7_SetPoint := 'True'} : ESTOP1;
   //    ESTOP_4 { S7_SetPoint := 'True'} : ESTOP1;
   //    TON_1 { ExternalWritable := 'False'} : TON;
   //    TON_2 { ExternalWritable := 'False'} : TON;
   //    TON_3 { ExternalWritable := 'False'} : TON;
   //    TON_4 { ExternalWritable := 'False'} : TON;
   // END_VAR
BEGIN
END_DATA_BLOCK

DATA_BLOCK "n0041-uc27-el001-k30001_SN51_2"   // DB1097, F_DB
VERSION : 0.1
// stored: AutoNumber true, DBAccessibleFromOPCUA true, DBAccessibleFromWebserver true, InstanceOfName 00_Push-Button_Input, InstanceOfType FB
"00_Push-Button_Input"
   // VAR_INPUT
   //    IN_1 : Bool;
   //    IN_2 : Bool;
   //    IN_3 : Bool;
   //    IN_4 : Bool;
   //    ON_Tristate : Bool;
   //    ON_Lamp : Bool;
   //    Reset : Bool;
   //    REAC_DELAY { ExternalWritable := 'False'} : Time;
   //    Bypass_ET200 : Bool;
   // END_VAR
   // VAR_OUTPUT
   //    OUT_1 : Bool;
   //    OUT_2 : Bool;
   //    OUT_3 : Bool;
   //    OUT_4 : Bool;
   //    Diag_1 : Bool;
   //    Diag_2 : Bool;
   //    Diag_3 : Bool;
   //    Diag_4 : Bool;
   //    Lamp_1 : Bool;
   //    Lamp_2 : Bool;
   //    Lamp_3 : Bool;
   //    Lamp_4 : Bool;
   // END_VAR
   // VAR
   //    ESTOP_1 { S7_SetPoint := 'True'} : ESTOP1;
   //    ESTOP_2 { S7_SetPoint := 'True'} : ESTOP1;
   //    ESTOP_3 { S7_SetPoint := 'True'} : ESTOP1;
   //    ESTOP_4 { S7_SetPoint := 'True'} : ESTOP1;
   //    TON_1 { ExternalWritable := 'False'} : TON;
   //    TON_2 { ExternalWritable := 'False'} : TON;
   //    TON_3 { ExternalWritable := 'False'} : TON;
   //    TON_4 { ExternalWritable := 'False'} : TON;
   // END_VAR
BEGIN
END_DATA_BLOCK

DATA_BLOCK "n0042-uc274-xn10_SN51_1"   // DB1098, F_DB
VERSION : 0.1
// stored: AutoNumber true, DBAccessibleFromOPCUA true, DBAccessibleFromWebserver true, InstanceOfName 00_Push-Button_Input, InstanceOfType FB
"00_Push-Button_Input"
   // VAR_INPUT
   //    IN_1 : Bool;
   //    IN_2 : Bool;
   //    IN_3 : Bool;
   //    IN_4 : Bool;
   //    ON_Tristate : Bool;
   //    ON_Lamp : Bool;
   //    Reset : Bool;
   //    REAC_DELAY { ExternalWritable := 'False'} : Time;
   //    Bypass_ET200 : Bool;
   // END_VAR
   // VAR_OUTPUT
   //    OUT_1 : Bool;
   //    OUT_2 : Bool;
   //    OUT_3 : Bool;
   //    OUT_4 : Bool;
   //    Diag_1 : Bool;
   //    Diag_2 : Bool;
   //    Diag_3 : Bool;
   //    Diag_4 : Bool;
   //    Lamp_1 : Bool;
   //    Lamp_2 : Bool;
   //    Lamp_3 : Bool;
   //    Lamp_4 : Bool;
   // END_VAR
   // VAR
   //    ESTOP_1 { S7_SetPoint := 'True'} : ESTOP1;
   //    ESTOP_2 { S7_SetPoint := 'True'} : ESTOP1;
   //    ESTOP_3 { S7_SetPoint := 'True'} : ESTOP1;
   //    ESTOP_4 { S7_SetPoint := 'True'} : ESTOP1;
   //    TON_1 { ExternalWritable := 'False'} : TON;
   //    TON_2 { ExternalWritable := 'False'} : TON;
   //    TON_3 { ExternalWritable := 'False'} : TON;
   //    TON_4 { ExternalWritable := 'False'} : TON;
   // END_VAR
BEGIN
END_DATA_BLOCK

DATA_BLOCK "n0042-uc274-xn10_SN51_2"   // DB1099, F_DB
VERSION : 0.1
// stored: AutoNumber true, DBAccessibleFromOPCUA true, DBAccessibleFromWebserver true, InstanceOfName 00_Push-Button_Input, InstanceOfType FB
"00_Push-Button_Input"
   // VAR_INPUT
   //    IN_1 : Bool;
   //    IN_2 : Bool;
   //    IN_3 : Bool;
   //    IN_4 : Bool;
   //    ON_Tristate : Bool;
   //    ON_Lamp : Bool;
   //    Reset : Bool;
   //    REAC_DELAY { ExternalWritable := 'False'} : Time;
   //    Bypass_ET200 : Bool;
   // END_VAR
   // VAR_OUTPUT
   //    OUT_1 : Bool;
   //    OUT_2 : Bool;
   //    OUT_3 : Bool;
   //    OUT_4 : Bool;
   //    Diag_1 : Bool;
   //    Diag_2 : Bool;
   //    Diag_3 : Bool;
   //    Diag_4 : Bool;
   //    Lamp_1 : Bool;
   //    Lamp_2 : Bool;
   //    Lamp_3 : Bool;
   //    Lamp_4 : Bool;
   // END_VAR
   // VAR
   //    ESTOP_1 { S7_SetPoint := 'True'} : ESTOP1;
   //    ESTOP_2 { S7_SetPoint := 'True'} : ESTOP1;
   //    ESTOP_3 { S7_SetPoint := 'True'} : ESTOP1;
   //    ESTOP_4 { S7_SetPoint := 'True'} : ESTOP1;
   //    TON_1 { ExternalWritable := 'False'} : TON;
   //    TON_2 { ExternalWritable := 'False'} : TON;
   //    TON_3 { ExternalWritable := 'False'} : TON;
   //    TON_4 { ExternalWritable := 'False'} : TON;
   // END_VAR
BEGIN
END_DATA_BLOCK

DATA_BLOCK "n0046-uc25-el001-k30001_SN51_1"   // DB1100, F_DB
VERSION : 0.1
// stored: AutoNumber true, DBAccessibleFromOPCUA true, DBAccessibleFromWebserver true, InstanceOfName 00_Push-Button_Input, InstanceOfType FB
"00_Push-Button_Input"
   // VAR_INPUT
   //    IN_1 : Bool;
   //    IN_2 : Bool;
   //    IN_3 : Bool;
   //    IN_4 : Bool;
   //    ON_Tristate : Bool;
   //    ON_Lamp : Bool;
   //    Reset : Bool;
   //    REAC_DELAY { ExternalWritable := 'False'} : Time;
   //    Bypass_ET200 : Bool;
   // END_VAR
   // VAR_OUTPUT
   //    OUT_1 : Bool;
   //    OUT_2 : Bool;
   //    OUT_3 : Bool;
   //    OUT_4 : Bool;
   //    Diag_1 : Bool;
   //    Diag_2 : Bool;
   //    Diag_3 : Bool;
   //    Diag_4 : Bool;
   //    Lamp_1 : Bool;
   //    Lamp_2 : Bool;
   //    Lamp_3 : Bool;
   //    Lamp_4 : Bool;
   // END_VAR
   // VAR
   //    ESTOP_1 { S7_SetPoint := 'True'} : ESTOP1;
   //    ESTOP_2 { S7_SetPoint := 'True'} : ESTOP1;
   //    ESTOP_3 { S7_SetPoint := 'True'} : ESTOP1;
   //    ESTOP_4 { S7_SetPoint := 'True'} : ESTOP1;
   //    TON_1 { ExternalWritable := 'False'} : TON;
   //    TON_2 { ExternalWritable := 'False'} : TON;
   //    TON_3 { ExternalWritable := 'False'} : TON;
   //    TON_4 { ExternalWritable := 'False'} : TON;
   // END_VAR
BEGIN
END_DATA_BLOCK

DATA_BLOCK "n0046-uc25-el001-k30001_SN51_2"   // DB1101, F_DB
VERSION : 0.1
// stored: AutoNumber true, DBAccessibleFromOPCUA true, DBAccessibleFromWebserver true, InstanceOfName 00_Push-Button_Input, InstanceOfType FB
"00_Push-Button_Input"
   // VAR_INPUT
   //    IN_1 : Bool;
   //    IN_2 : Bool;
   //    IN_3 : Bool;
   //    IN_4 : Bool;
   //    ON_Tristate : Bool;
   //    ON_Lamp : Bool;
   //    Reset : Bool;
   //    REAC_DELAY { ExternalWritable := 'False'} : Time;
   //    Bypass_ET200 : Bool;
   // END_VAR
   // VAR_OUTPUT
   //    OUT_1 : Bool;
   //    OUT_2 : Bool;
   //    OUT_3 : Bool;
   //    OUT_4 : Bool;
   //    Diag_1 : Bool;
   //    Diag_2 : Bool;
   //    Diag_3 : Bool;
   //    Diag_4 : Bool;
   //    Lamp_1 : Bool;
   //    Lamp_2 : Bool;
   //    Lamp_3 : Bool;
   //    Lamp_4 : Bool;
   // END_VAR
   // VAR
   //    ESTOP_1 { S7_SetPoint := 'True'} : ESTOP1;
   //    ESTOP_2 { S7_SetPoint := 'True'} : ESTOP1;
   //    ESTOP_3 { S7_SetPoint := 'True'} : ESTOP1;
   //    ESTOP_4 { S7_SetPoint := 'True'} : ESTOP1;
   //    TON_1 { ExternalWritable := 'False'} : TON;
   //    TON_2 { ExternalWritable := 'False'} : TON;
   //    TON_3 { ExternalWritable := 'False'} : TON;
   //    TON_4 { ExternalWritable := 'False'} : TON;
   // END_VAR
BEGIN
END_DATA_BLOCK

DATA_BLOCK "n0046-uc25-el001-k30001_SN51_3"   // DB1102, F_DB
VERSION : 0.1
// stored: AutoNumber true, DBAccessibleFromOPCUA true, DBAccessibleFromWebserver true, InstanceOfName 00_Push-Button_Input, InstanceOfType FB
"00_Push-Button_Input"
   // VAR_INPUT
   //    IN_1 : Bool;
   //    IN_2 : Bool;
   //    IN_3 : Bool;
   //    IN_4 : Bool;
   //    ON_Tristate : Bool;
   //    ON_Lamp : Bool;
   //    Reset : Bool;
   //    REAC_DELAY { ExternalWritable := 'False'} : Time;
   //    Bypass_ET200 : Bool;
   // END_VAR
   // VAR_OUTPUT
   //    OUT_1 : Bool;
   //    OUT_2 : Bool;
   //    OUT_3 : Bool;
   //    OUT_4 : Bool;
   //    Diag_1 : Bool;
   //    Diag_2 : Bool;
   //    Diag_3 : Bool;
   //    Diag_4 : Bool;
   //    Lamp_1 : Bool;
   //    Lamp_2 : Bool;
   //    Lamp_3 : Bool;
   //    Lamp_4 : Bool;
   // END_VAR
   // VAR
   //    ESTOP_1 { S7_SetPoint := 'True'} : ESTOP1;
   //    ESTOP_2 { S7_SetPoint := 'True'} : ESTOP1;
   //    ESTOP_3 { S7_SetPoint := 'True'} : ESTOP1;
   //    ESTOP_4 { S7_SetPoint := 'True'} : ESTOP1;
   //    TON_1 { ExternalWritable := 'False'} : TON;
   //    TON_2 { ExternalWritable := 'False'} : TON;
   //    TON_3 { ExternalWritable := 'False'} : TON;
   //    TON_4 { ExternalWritable := 'False'} : TON;
   // END_VAR
BEGIN
END_DATA_BLOCK

DATA_BLOCK "n0047-uc254-xn10_SN51_1"   // DB1103, F_DB
VERSION : 0.1
// stored: AutoNumber true, DBAccessibleFromOPCUA true, DBAccessibleFromWebserver true, InstanceOfName 00_Push-Button_Input, InstanceOfType FB
"00_Push-Button_Input"
   // VAR_INPUT
   //    IN_1 : Bool;
   //    IN_2 : Bool;
   //    IN_3 : Bool;
   //    IN_4 : Bool;
   //    ON_Tristate : Bool;
   //    ON_Lamp : Bool;
   //    Reset : Bool;
   //    REAC_DELAY { ExternalWritable := 'False'} : Time;
   //    Bypass_ET200 : Bool;
   // END_VAR
   // VAR_OUTPUT
   //    OUT_1 : Bool;
   //    OUT_2 : Bool;
   //    OUT_3 : Bool;
   //    OUT_4 : Bool;
   //    Diag_1 : Bool;
   //    Diag_2 : Bool;
   //    Diag_3 : Bool;
   //    Diag_4 : Bool;
   //    Lamp_1 : Bool;
   //    Lamp_2 : Bool;
   //    Lamp_3 : Bool;
   //    Lamp_4 : Bool;
   // END_VAR
   // VAR
   //    ESTOP_1 { S7_SetPoint := 'True'} : ESTOP1;
   //    ESTOP_2 { S7_SetPoint := 'True'} : ESTOP1;
   //    ESTOP_3 { S7_SetPoint := 'True'} : ESTOP1;
   //    ESTOP_4 { S7_SetPoint := 'True'} : ESTOP1;
   //    TON_1 { ExternalWritable := 'False'} : TON;
   //    TON_2 { ExternalWritable := 'False'} : TON;
   //    TON_3 { ExternalWritable := 'False'} : TON;
   //    TON_4 { ExternalWritable := 'False'} : TON;
   // END_VAR
BEGIN
END_DATA_BLOCK

DATA_BLOCK "n0047-uc254-xn10_SN51_2"   // DB1104, F_DB
VERSION : 0.1
// stored: AutoNumber true, DBAccessibleFromOPCUA true, DBAccessibleFromWebserver true, InstanceOfName 00_Push-Button_Input, InstanceOfType FB
"00_Push-Button_Input"
   // VAR_INPUT
   //    IN_1 : Bool;
   //    IN_2 : Bool;
   //    IN_3 : Bool;
   //    IN_4 : Bool;
   //    ON_Tristate : Bool;
   //    ON_Lamp : Bool;
   //    Reset : Bool;
   //    REAC_DELAY { ExternalWritable := 'False'} : Time;
   //    Bypass_ET200 : Bool;
   // END_VAR
   // VAR_OUTPUT
   //    OUT_1 : Bool;
   //    OUT_2 : Bool;
   //    OUT_3 : Bool;
   //    OUT_4 : Bool;
   //    Diag_1 : Bool;
   //    Diag_2 : Bool;
   //    Diag_3 : Bool;
   //    Diag_4 : Bool;
   //    Lamp_1 : Bool;
   //    Lamp_2 : Bool;
   //    Lamp_3 : Bool;
   //    Lamp_4 : Bool;
   // END_VAR
   // VAR
   //    ESTOP_1 { S7_SetPoint := 'True'} : ESTOP1;
   //    ESTOP_2 { S7_SetPoint := 'True'} : ESTOP1;
   //    ESTOP_3 { S7_SetPoint := 'True'} : ESTOP1;
   //    ESTOP_4 { S7_SetPoint := 'True'} : ESTOP1;
   //    TON_1 { ExternalWritable := 'False'} : TON;
   //    TON_2 { ExternalWritable := 'False'} : TON;
   //    TON_3 { ExternalWritable := 'False'} : TON;
   //    TON_4 { ExternalWritable := 'False'} : TON;
   // END_VAR
BEGIN
END_DATA_BLOCK

DATA_BLOCK "n0051-uc24-el001-k30001_SN51_1"   // DB1105, F_DB
VERSION : 0.1
// stored: AutoNumber true, DBAccessibleFromOPCUA true, DBAccessibleFromWebserver true, InstanceOfName 00_Push-Button_Input, InstanceOfType FB
"00_Push-Button_Input"
   // VAR_INPUT
   //    IN_1 : Bool;
   //    IN_2 : Bool;
   //    IN_3 : Bool;
   //    IN_4 : Bool;
   //    ON_Tristate : Bool;
   //    ON_Lamp : Bool;
   //    Reset : Bool;
   //    REAC_DELAY { ExternalWritable := 'False'} : Time;
   //    Bypass_ET200 : Bool;
   // END_VAR
   // VAR_OUTPUT
   //    OUT_1 : Bool;
   //    OUT_2 : Bool;
   //    OUT_3 : Bool;
   //    OUT_4 : Bool;
   //    Diag_1 : Bool;
   //    Diag_2 : Bool;
   //    Diag_3 : Bool;
   //    Diag_4 : Bool;
   //    Lamp_1 : Bool;
   //    Lamp_2 : Bool;
   //    Lamp_3 : Bool;
   //    Lamp_4 : Bool;
   // END_VAR
   // VAR
   //    ESTOP_1 { S7_SetPoint := 'True'} : ESTOP1;
   //    ESTOP_2 { S7_SetPoint := 'True'} : ESTOP1;
   //    ESTOP_3 { S7_SetPoint := 'True'} : ESTOP1;
   //    ESTOP_4 { S7_SetPoint := 'True'} : ESTOP1;
   //    TON_1 { ExternalWritable := 'False'} : TON;
   //    TON_2 { ExternalWritable := 'False'} : TON;
   //    TON_3 { ExternalWritable := 'False'} : TON;
   //    TON_4 { ExternalWritable := 'False'} : TON;
   // END_VAR
BEGIN
END_DATA_BLOCK

DATA_BLOCK "n0051-uc24-el001-k30001_SN51_2"   // DB1106, F_DB
VERSION : 0.1
// stored: AutoNumber true, DBAccessibleFromOPCUA true, DBAccessibleFromWebserver true, InstanceOfName 00_Push-Button_Input, InstanceOfType FB
"00_Push-Button_Input"
   // VAR_INPUT
   //    IN_1 : Bool;
   //    IN_2 : Bool;
   //    IN_3 : Bool;
   //    IN_4 : Bool;
   //    ON_Tristate : Bool;
   //    ON_Lamp : Bool;
   //    Reset : Bool;
   //    REAC_DELAY { ExternalWritable := 'False'} : Time;
   //    Bypass_ET200 : Bool;
   // END_VAR
   // VAR_OUTPUT
   //    OUT_1 : Bool;
   //    OUT_2 : Bool;
   //    OUT_3 : Bool;
   //    OUT_4 : Bool;
   //    Diag_1 : Bool;
   //    Diag_2 : Bool;
   //    Diag_3 : Bool;
   //    Diag_4 : Bool;
   //    Lamp_1 : Bool;
   //    Lamp_2 : Bool;
   //    Lamp_3 : Bool;
   //    Lamp_4 : Bool;
   // END_VAR
   // VAR
   //    ESTOP_1 { S7_SetPoint := 'True'} : ESTOP1;
   //    ESTOP_2 { S7_SetPoint := 'True'} : ESTOP1;
   //    ESTOP_3 { S7_SetPoint := 'True'} : ESTOP1;
   //    ESTOP_4 { S7_SetPoint := 'True'} : ESTOP1;
   //    TON_1 { ExternalWritable := 'False'} : TON;
   //    TON_2 { ExternalWritable := 'False'} : TON;
   //    TON_3 { ExternalWritable := 'False'} : TON;
   //    TON_4 { ExternalWritable := 'False'} : TON;
   // END_VAR
BEGIN
END_DATA_BLOCK

DATA_BLOCK "n0051-uc24-el001-k30001_SN51_3"   // DB1107, F_DB
VERSION : 0.1
// stored: AutoNumber true, DBAccessibleFromOPCUA true, DBAccessibleFromWebserver true, InstanceOfName 00_Push-Button_Input, InstanceOfType FB
"00_Push-Button_Input"
   // VAR_INPUT
   //    IN_1 : Bool;
   //    IN_2 : Bool;
   //    IN_3 : Bool;
   //    IN_4 : Bool;
   //    ON_Tristate : Bool;
   //    ON_Lamp : Bool;
   //    Reset : Bool;
   //    REAC_DELAY { ExternalWritable := 'False'} : Time;
   //    Bypass_ET200 : Bool;
   // END_VAR
   // VAR_OUTPUT
   //    OUT_1 : Bool;
   //    OUT_2 : Bool;
   //    OUT_3 : Bool;
   //    OUT_4 : Bool;
   //    Diag_1 : Bool;
   //    Diag_2 : Bool;
   //    Diag_3 : Bool;
   //    Diag_4 : Bool;
   //    Lamp_1 : Bool;
   //    Lamp_2 : Bool;
   //    Lamp_3 : Bool;
   //    Lamp_4 : Bool;
   // END_VAR
   // VAR
   //    ESTOP_1 { S7_SetPoint := 'True'} : ESTOP1;
   //    ESTOP_2 { S7_SetPoint := 'True'} : ESTOP1;
   //    ESTOP_3 { S7_SetPoint := 'True'} : ESTOP1;
   //    ESTOP_4 { S7_SetPoint := 'True'} : ESTOP1;
   //    TON_1 { ExternalWritable := 'False'} : TON;
   //    TON_2 { ExternalWritable := 'False'} : TON;
   //    TON_3 { ExternalWritable := 'False'} : TON;
   //    TON_4 { ExternalWritable := 'False'} : TON;
   // END_VAR
BEGIN
END_DATA_BLOCK

DATA_BLOCK "n0052-uc244-xn10_SN51_1"   // DB1108, F_DB
VERSION : 0.1
// stored: AutoNumber true, DBAccessibleFromOPCUA true, DBAccessibleFromWebserver true, InstanceOfName 00_Push-Button_Input, InstanceOfType FB
"00_Push-Button_Input"
   // VAR_INPUT
   //    IN_1 : Bool;
   //    IN_2 : Bool;
   //    IN_3 : Bool;
   //    IN_4 : Bool;
   //    ON_Tristate : Bool;
   //    ON_Lamp : Bool;
   //    Reset : Bool;
   //    REAC_DELAY { ExternalWritable := 'False'} : Time;
   //    Bypass_ET200 : Bool;
   // END_VAR
   // VAR_OUTPUT
   //    OUT_1 : Bool;
   //    OUT_2 : Bool;
   //    OUT_3 : Bool;
   //    OUT_4 : Bool;
   //    Diag_1 : Bool;
   //    Diag_2 : Bool;
   //    Diag_3 : Bool;
   //    Diag_4 : Bool;
   //    Lamp_1 : Bool;
   //    Lamp_2 : Bool;
   //    Lamp_3 : Bool;
   //    Lamp_4 : Bool;
   // END_VAR
   // VAR
   //    ESTOP_1 { S7_SetPoint := 'True'} : ESTOP1;
   //    ESTOP_2 { S7_SetPoint := 'True'} : ESTOP1;
   //    ESTOP_3 { S7_SetPoint := 'True'} : ESTOP1;
   //    ESTOP_4 { S7_SetPoint := 'True'} : ESTOP1;
   //    TON_1 { ExternalWritable := 'False'} : TON;
   //    TON_2 { ExternalWritable := 'False'} : TON;
   //    TON_3 { ExternalWritable := 'False'} : TON;
   //    TON_4 { ExternalWritable := 'False'} : TON;
   // END_VAR
BEGIN
END_DATA_BLOCK

DATA_BLOCK "n0052-uc244-xn10_SN51_2"   // DB1109, F_DB
VERSION : 0.1
// stored: AutoNumber true, DBAccessibleFromOPCUA true, DBAccessibleFromWebserver true, InstanceOfName 00_Push-Button_Input, InstanceOfType FB
"00_Push-Button_Input"
   // VAR_INPUT
   //    IN_1 : Bool;
   //    IN_2 : Bool;
   //    IN_3 : Bool;
   //    IN_4 : Bool;
   //    ON_Tristate : Bool;
   //    ON_Lamp : Bool;
   //    Reset : Bool;
   //    REAC_DELAY { ExternalWritable := 'False'} : Time;
   //    Bypass_ET200 : Bool;
   // END_VAR
   // VAR_OUTPUT
   //    OUT_1 : Bool;
   //    OUT_2 : Bool;
   //    OUT_3 : Bool;
   //    OUT_4 : Bool;
   //    Diag_1 : Bool;
   //    Diag_2 : Bool;
   //    Diag_3 : Bool;
   //    Diag_4 : Bool;
   //    Lamp_1 : Bool;
   //    Lamp_2 : Bool;
   //    Lamp_3 : Bool;
   //    Lamp_4 : Bool;
   // END_VAR
   // VAR
   //    ESTOP_1 { S7_SetPoint := 'True'} : ESTOP1;
   //    ESTOP_2 { S7_SetPoint := 'True'} : ESTOP1;
   //    ESTOP_3 { S7_SetPoint := 'True'} : ESTOP1;
   //    ESTOP_4 { S7_SetPoint := 'True'} : ESTOP1;
   //    TON_1 { ExternalWritable := 'False'} : TON;
   //    TON_2 { ExternalWritable := 'False'} : TON;
   //    TON_3 { ExternalWritable := 'False'} : TON;
   //    TON_4 { ExternalWritable := 'False'} : TON;
   // END_VAR
BEGIN
END_DATA_BLOCK

DATA_BLOCK "n0056-uc23-el001-k30001_SN51_1"   // DB1110, F_DB
VERSION : 0.1
// stored: AutoNumber true, DBAccessibleFromOPCUA true, DBAccessibleFromWebserver true, InstanceOfName 00_Push-Button_Input, InstanceOfType FB
"00_Push-Button_Input"
   // VAR_INPUT
   //    IN_1 : Bool;
   //    IN_2 : Bool;
   //    IN_3 : Bool;
   //    IN_4 : Bool;
   //    ON_Tristate : Bool;
   //    ON_Lamp : Bool;
   //    Reset : Bool;
   //    REAC_DELAY { ExternalWritable := 'False'} : Time;
   //    Bypass_ET200 : Bool;
   // END_VAR
   // VAR_OUTPUT
   //    OUT_1 : Bool;
   //    OUT_2 : Bool;
   //    OUT_3 : Bool;
   //    OUT_4 : Bool;
   //    Diag_1 : Bool;
   //    Diag_2 : Bool;
   //    Diag_3 : Bool;
   //    Diag_4 : Bool;
   //    Lamp_1 : Bool;
   //    Lamp_2 : Bool;
   //    Lamp_3 : Bool;
   //    Lamp_4 : Bool;
   // END_VAR
   // VAR
   //    ESTOP_1 { S7_SetPoint := 'True'} : ESTOP1;
   //    ESTOP_2 { S7_SetPoint := 'True'} : ESTOP1;
   //    ESTOP_3 { S7_SetPoint := 'True'} : ESTOP1;
   //    ESTOP_4 { S7_SetPoint := 'True'} : ESTOP1;
   //    TON_1 { ExternalWritable := 'False'} : TON;
   //    TON_2 { ExternalWritable := 'False'} : TON;
   //    TON_3 { ExternalWritable := 'False'} : TON;
   //    TON_4 { ExternalWritable := 'False'} : TON;
   // END_VAR
BEGIN
END_DATA_BLOCK

DATA_BLOCK "n0056-uc23-el001-k30001_SN51_2"   // DB1111, F_DB
VERSION : 0.1
// stored: AutoNumber true, DBAccessibleFromOPCUA true, DBAccessibleFromWebserver true, InstanceOfName 00_Push-Button_Input, InstanceOfType FB
"00_Push-Button_Input"
   // VAR_INPUT
   //    IN_1 : Bool;
   //    IN_2 : Bool;
   //    IN_3 : Bool;
   //    IN_4 : Bool;
   //    ON_Tristate : Bool;
   //    ON_Lamp : Bool;
   //    Reset : Bool;
   //    REAC_DELAY { ExternalWritable := 'False'} : Time;
   //    Bypass_ET200 : Bool;
   // END_VAR
   // VAR_OUTPUT
   //    OUT_1 : Bool;
   //    OUT_2 : Bool;
   //    OUT_3 : Bool;
   //    OUT_4 : Bool;
   //    Diag_1 : Bool;
   //    Diag_2 : Bool;
   //    Diag_3 : Bool;
   //    Diag_4 : Bool;
   //    Lamp_1 : Bool;
   //    Lamp_2 : Bool;
   //    Lamp_3 : Bool;
   //    Lamp_4 : Bool;
   // END_VAR
   // VAR
   //    ESTOP_1 { S7_SetPoint := 'True'} : ESTOP1;
   //    ESTOP_2 { S7_SetPoint := 'True'} : ESTOP1;
   //    ESTOP_3 { S7_SetPoint := 'True'} : ESTOP1;
   //    ESTOP_4 { S7_SetPoint := 'True'} : ESTOP1;
   //    TON_1 { ExternalWritable := 'False'} : TON;
   //    TON_2 { ExternalWritable := 'False'} : TON;
   //    TON_3 { ExternalWritable := 'False'} : TON;
   //    TON_4 { ExternalWritable := 'False'} : TON;
   // END_VAR
BEGIN
END_DATA_BLOCK

DATA_BLOCK "n0056-uc23-el001-k30001_SN51_3"   // DB1112, F_DB
VERSION : 0.1
// stored: AutoNumber true, DBAccessibleFromOPCUA true, DBAccessibleFromWebserver true, InstanceOfName 00_Push-Button_Input, InstanceOfType FB
"00_Push-Button_Input"
   // VAR_INPUT
   //    IN_1 : Bool;
   //    IN_2 : Bool;
   //    IN_3 : Bool;
   //    IN_4 : Bool;
   //    ON_Tristate : Bool;
   //    ON_Lamp : Bool;
   //    Reset : Bool;
   //    REAC_DELAY { ExternalWritable := 'False'} : Time;
   //    Bypass_ET200 : Bool;
   // END_VAR
   // VAR_OUTPUT
   //    OUT_1 : Bool;
   //    OUT_2 : Bool;
   //    OUT_3 : Bool;
   //    OUT_4 : Bool;
   //    Diag_1 : Bool;
   //    Diag_2 : Bool;
   //    Diag_3 : Bool;
   //    Diag_4 : Bool;
   //    Lamp_1 : Bool;
   //    Lamp_2 : Bool;
   //    Lamp_3 : Bool;
   //    Lamp_4 : Bool;
   // END_VAR
   // VAR
   //    ESTOP_1 { S7_SetPoint := 'True'} : ESTOP1;
   //    ESTOP_2 { S7_SetPoint := 'True'} : ESTOP1;
   //    ESTOP_3 { S7_SetPoint := 'True'} : ESTOP1;
   //    ESTOP_4 { S7_SetPoint := 'True'} : ESTOP1;
   //    TON_1 { ExternalWritable := 'False'} : TON;
   //    TON_2 { ExternalWritable := 'False'} : TON;
   //    TON_3 { ExternalWritable := 'False'} : TON;
   //    TON_4 { ExternalWritable := 'False'} : TON;
   // END_VAR
BEGIN
END_DATA_BLOCK

DATA_BLOCK "n0057-uc234-xn10_SN51_1"   // DB1113, F_DB
VERSION : 0.1
// stored: AutoNumber true, DBAccessibleFromOPCUA true, DBAccessibleFromWebserver true, InstanceOfName 00_Push-Button_Input, InstanceOfType FB
"00_Push-Button_Input"
   // VAR_INPUT
   //    IN_1 : Bool;
   //    IN_2 : Bool;
   //    IN_3 : Bool;
   //    IN_4 : Bool;
   //    ON_Tristate : Bool;
   //    ON_Lamp : Bool;
   //    Reset : Bool;
   //    REAC_DELAY { ExternalWritable := 'False'} : Time;
   //    Bypass_ET200 : Bool;
   // END_VAR
   // VAR_OUTPUT
   //    OUT_1 : Bool;
   //    OUT_2 : Bool;
   //    OUT_3 : Bool;
   //    OUT_4 : Bool;
   //    Diag_1 : Bool;
   //    Diag_2 : Bool;
   //    Diag_3 : Bool;
   //    Diag_4 : Bool;
   //    Lamp_1 : Bool;
   //    Lamp_2 : Bool;
   //    Lamp_3 : Bool;
   //    Lamp_4 : Bool;
   // END_VAR
   // VAR
   //    ESTOP_1 { S7_SetPoint := 'True'} : ESTOP1;
   //    ESTOP_2 { S7_SetPoint := 'True'} : ESTOP1;
   //    ESTOP_3 { S7_SetPoint := 'True'} : ESTOP1;
   //    ESTOP_4 { S7_SetPoint := 'True'} : ESTOP1;
   //    TON_1 { ExternalWritable := 'False'} : TON;
   //    TON_2 { ExternalWritable := 'False'} : TON;
   //    TON_3 { ExternalWritable := 'False'} : TON;
   //    TON_4 { ExternalWritable := 'False'} : TON;
   // END_VAR
BEGIN
END_DATA_BLOCK

DATA_BLOCK "n0057-uc234-xn10_SN51_2"   // DB1114, F_DB
VERSION : 0.1
// stored: AutoNumber true, DBAccessibleFromOPCUA true, DBAccessibleFromWebserver true, InstanceOfName 00_Push-Button_Input, InstanceOfType FB
"00_Push-Button_Input"
   // VAR_INPUT
   //    IN_1 : Bool;
   //    IN_2 : Bool;
   //    IN_3 : Bool;
   //    IN_4 : Bool;
   //    ON_Tristate : Bool;
   //    ON_Lamp : Bool;
   //    Reset : Bool;
   //    REAC_DELAY { ExternalWritable := 'False'} : Time;
   //    Bypass_ET200 : Bool;
   // END_VAR
   // VAR_OUTPUT
   //    OUT_1 : Bool;
   //    OUT_2 : Bool;
   //    OUT_3 : Bool;
   //    OUT_4 : Bool;
   //    Diag_1 : Bool;
   //    Diag_2 : Bool;
   //    Diag_3 : Bool;
   //    Diag_4 : Bool;
   //    Lamp_1 : Bool;
   //    Lamp_2 : Bool;
   //    Lamp_3 : Bool;
   //    Lamp_4 : Bool;
   // END_VAR
   // VAR
   //    ESTOP_1 { S7_SetPoint := 'True'} : ESTOP1;
   //    ESTOP_2 { S7_SetPoint := 'True'} : ESTOP1;
   //    ESTOP_3 { S7_SetPoint := 'True'} : ESTOP1;
   //    ESTOP_4 { S7_SetPoint := 'True'} : ESTOP1;
   //    TON_1 { ExternalWritable := 'False'} : TON;
   //    TON_2 { ExternalWritable := 'False'} : TON;
   //    TON_3 { ExternalWritable := 'False'} : TON;
   //    TON_4 { ExternalWritable := 'False'} : TON;
   // END_VAR
BEGIN
END_DATA_BLOCK

DATA_BLOCK "n0058-ct2-el003-k30001_SN51_1"   // DB1115, F_DB
VERSION : 0.1
// stored: AutoNumber true, DBAccessibleFromOPCUA true, DBAccessibleFromWebserver true, InstanceOfName 00_Push-Button_Input, InstanceOfType FB
"00_Push-Button_Input"
   // VAR_INPUT
   //    IN_1 : Bool;
   //    IN_2 : Bool;
   //    IN_3 : Bool;
   //    IN_4 : Bool;
   //    ON_Tristate : Bool;
   //    ON_Lamp : Bool;
   //    Reset : Bool;
   //    REAC_DELAY { ExternalWritable := 'False'} : Time;
   //    Bypass_ET200 : Bool;
   // END_VAR
   // VAR_OUTPUT
   //    OUT_1 : Bool;
   //    OUT_2 : Bool;
   //    OUT_3 : Bool;
   //    OUT_4 : Bool;
   //    Diag_1 : Bool;
   //    Diag_2 : Bool;
   //    Diag_3 : Bool;
   //    Diag_4 : Bool;
   //    Lamp_1 : Bool;
   //    Lamp_2 : Bool;
   //    Lamp_3 : Bool;
   //    Lamp_4 : Bool;
   // END_VAR
   // VAR
   //    ESTOP_1 { S7_SetPoint := 'True'} : ESTOP1;
   //    ESTOP_2 { S7_SetPoint := 'True'} : ESTOP1;
   //    ESTOP_3 { S7_SetPoint := 'True'} : ESTOP1;
   //    ESTOP_4 { S7_SetPoint := 'True'} : ESTOP1;
   //    TON_1 { ExternalWritable := 'False'} : TON;
   //    TON_2 { ExternalWritable := 'False'} : TON;
   //    TON_3 { ExternalWritable := 'False'} : TON;
   //    TON_4 { ExternalWritable := 'False'} : TON;
   // END_VAR
BEGIN
END_DATA_BLOCK

DATA_BLOCK "n0058-ct2-el003-k30001_SN51_2"   // DB1116, F_DB
VERSION : 0.1
// stored: AutoNumber true, DBAccessibleFromOPCUA true, DBAccessibleFromWebserver true, InstanceOfName 00_Push-Button_Input, InstanceOfType FB
"00_Push-Button_Input"
   // VAR_INPUT
   //    IN_1 : Bool;
   //    IN_2 : Bool;
   //    IN_3 : Bool;
   //    IN_4 : Bool;
   //    ON_Tristate : Bool;
   //    ON_Lamp : Bool;
   //    Reset : Bool;
   //    REAC_DELAY { ExternalWritable := 'False'} : Time;
   //    Bypass_ET200 : Bool;
   // END_VAR
   // VAR_OUTPUT
   //    OUT_1 : Bool;
   //    OUT_2 : Bool;
   //    OUT_3 : Bool;
   //    OUT_4 : Bool;
   //    Diag_1 : Bool;
   //    Diag_2 : Bool;
   //    Diag_3 : Bool;
   //    Diag_4 : Bool;
   //    Lamp_1 : Bool;
   //    Lamp_2 : Bool;
   //    Lamp_3 : Bool;
   //    Lamp_4 : Bool;
   // END_VAR
   // VAR
   //    ESTOP_1 { S7_SetPoint := 'True'} : ESTOP1;
   //    ESTOP_2 { S7_SetPoint := 'True'} : ESTOP1;
   //    ESTOP_3 { S7_SetPoint := 'True'} : ESTOP1;
   //    ESTOP_4 { S7_SetPoint := 'True'} : ESTOP1;
   //    TON_1 { ExternalWritable := 'False'} : TON;
   //    TON_2 { ExternalWritable := 'False'} : TON;
   //    TON_3 { ExternalWritable := 'False'} : TON;
   //    TON_4 { ExternalWritable := 'False'} : TON;
   // END_VAR
BEGIN
END_DATA_BLOCK

DATA_BLOCK "n0058-ct2-el003-k30001_SN51_3"   // DB1117, F_DB
VERSION : 0.1
// stored: AutoNumber true, DBAccessibleFromOPCUA true, DBAccessibleFromWebserver true, InstanceOfName 00_Push-Button_Input, InstanceOfType FB
"00_Push-Button_Input"
   // VAR_INPUT
   //    IN_1 : Bool;
   //    IN_2 : Bool;
   //    IN_3 : Bool;
   //    IN_4 : Bool;
   //    ON_Tristate : Bool;
   //    ON_Lamp : Bool;
   //    Reset : Bool;
   //    REAC_DELAY { ExternalWritable := 'False'} : Time;
   //    Bypass_ET200 : Bool;
   // END_VAR
   // VAR_OUTPUT
   //    OUT_1 : Bool;
   //    OUT_2 : Bool;
   //    OUT_3 : Bool;
   //    OUT_4 : Bool;
   //    Diag_1 : Bool;
   //    Diag_2 : Bool;
   //    Diag_3 : Bool;
   //    Diag_4 : Bool;
   //    Lamp_1 : Bool;
   //    Lamp_2 : Bool;
   //    Lamp_3 : Bool;
   //    Lamp_4 : Bool;
   // END_VAR
   // VAR
   //    ESTOP_1 { S7_SetPoint := 'True'} : ESTOP1;
   //    ESTOP_2 { S7_SetPoint := 'True'} : ESTOP1;
   //    ESTOP_3 { S7_SetPoint := 'True'} : ESTOP1;
   //    ESTOP_4 { S7_SetPoint := 'True'} : ESTOP1;
   //    TON_1 { ExternalWritable := 'False'} : TON;
   //    TON_2 { ExternalWritable := 'False'} : TON;
   //    TON_3 { ExternalWritable := 'False'} : TON;
   //    TON_4 { ExternalWritable := 'False'} : TON;
   // END_VAR
BEGIN
END_DATA_BLOCK

DATA_BLOCK "n0058-ct2-el003-k30001_SN51_4"   // DB1118, F_DB
VERSION : 0.1
// stored: AutoNumber true, DBAccessibleFromOPCUA true, DBAccessibleFromWebserver true, InstanceOfName 00_Push-Button_Input, InstanceOfType FB
"00_Push-Button_Input"
   // VAR_INPUT
   //    IN_1 : Bool;
   //    IN_2 : Bool;
   //    IN_3 : Bool;
   //    IN_4 : Bool;
   //    ON_Tristate : Bool;
   //    ON_Lamp : Bool;
   //    Reset : Bool;
   //    REAC_DELAY { ExternalWritable := 'False'} : Time;
   //    Bypass_ET200 : Bool;
   // END_VAR
   // VAR_OUTPUT
   //    OUT_1 : Bool;
   //    OUT_2 : Bool;
   //    OUT_3 : Bool;
   //    OUT_4 : Bool;
   //    Diag_1 : Bool;
   //    Diag_2 : Bool;
   //    Diag_3 : Bool;
   //    Diag_4 : Bool;
   //    Lamp_1 : Bool;
   //    Lamp_2 : Bool;
   //    Lamp_3 : Bool;
   //    Lamp_4 : Bool;
   // END_VAR
   // VAR
   //    ESTOP_1 { S7_SetPoint := 'True'} : ESTOP1;
   //    ESTOP_2 { S7_SetPoint := 'True'} : ESTOP1;
   //    ESTOP_3 { S7_SetPoint := 'True'} : ESTOP1;
   //    ESTOP_4 { S7_SetPoint := 'True'} : ESTOP1;
   //    TON_1 { ExternalWritable := 'False'} : TON;
   //    TON_2 { ExternalWritable := 'False'} : TON;
   //    TON_3 { ExternalWritable := 'False'} : TON;
   //    TON_4 { ExternalWritable := 'False'} : TON;
   // END_VAR
BEGIN
END_DATA_BLOCK

DATA_BLOCK "n0058-ct2-el003-k30001_SN51_5"   // DB1119, F_DB
VERSION : 0.1
// stored: AutoNumber true, DBAccessibleFromOPCUA true, DBAccessibleFromWebserver true, InstanceOfName 00_Push-Button_Input, InstanceOfType FB
"00_Push-Button_Input"
   // VAR_INPUT
   //    IN_1 : Bool;
   //    IN_2 : Bool;
   //    IN_3 : Bool;
   //    IN_4 : Bool;
   //    ON_Tristate : Bool;
   //    ON_Lamp : Bool;
   //    Reset : Bool;
   //    REAC_DELAY { ExternalWritable := 'False'} : Time;
   //    Bypass_ET200 : Bool;
   // END_VAR
   // VAR_OUTPUT
   //    OUT_1 : Bool;
   //    OUT_2 : Bool;
   //    OUT_3 : Bool;
   //    OUT_4 : Bool;
   //    Diag_1 : Bool;
   //    Diag_2 : Bool;
   //    Diag_3 : Bool;
   //    Diag_4 : Bool;
   //    Lamp_1 : Bool;
   //    Lamp_2 : Bool;
   //    Lamp_3 : Bool;
   //    Lamp_4 : Bool;
   // END_VAR
   // VAR
   //    ESTOP_1 { S7_SetPoint := 'True'} : ESTOP1;
   //    ESTOP_2 { S7_SetPoint := 'True'} : ESTOP1;
   //    ESTOP_3 { S7_SetPoint := 'True'} : ESTOP1;
   //    ESTOP_4 { S7_SetPoint := 'True'} : ESTOP1;
   //    TON_1 { ExternalWritable := 'False'} : TON;
   //    TON_2 { ExternalWritable := 'False'} : TON;
   //    TON_3 { ExternalWritable := 'False'} : TON;
   //    TON_4 { ExternalWritable := 'False'} : TON;
   // END_VAR
BEGIN
END_DATA_BLOCK

DATA_BLOCK "n0061-uc22-el001-k30001_SN51_1"   // DB1120, F_DB
VERSION : 0.1
// stored: AutoNumber true, DBAccessibleFromOPCUA true, DBAccessibleFromWebserver true, InstanceOfName 00_Push-Button_Input, InstanceOfType FB
"00_Push-Button_Input"
   // VAR_INPUT
   //    IN_1 : Bool;
   //    IN_2 : Bool;
   //    IN_3 : Bool;
   //    IN_4 : Bool;
   //    ON_Tristate : Bool;
   //    ON_Lamp : Bool;
   //    Reset : Bool;
   //    REAC_DELAY { ExternalWritable := 'False'} : Time;
   //    Bypass_ET200 : Bool;
   // END_VAR
   // VAR_OUTPUT
   //    OUT_1 : Bool;
   //    OUT_2 : Bool;
   //    OUT_3 : Bool;
   //    OUT_4 : Bool;
   //    Diag_1 : Bool;
   //    Diag_2 : Bool;
   //    Diag_3 : Bool;
   //    Diag_4 : Bool;
   //    Lamp_1 : Bool;
   //    Lamp_2 : Bool;
   //    Lamp_3 : Bool;
   //    Lamp_4 : Bool;
   // END_VAR
   // VAR
   //    ESTOP_1 { S7_SetPoint := 'True'} : ESTOP1;
   //    ESTOP_2 { S7_SetPoint := 'True'} : ESTOP1;
   //    ESTOP_3 { S7_SetPoint := 'True'} : ESTOP1;
   //    ESTOP_4 { S7_SetPoint := 'True'} : ESTOP1;
   //    TON_1 { ExternalWritable := 'False'} : TON;
   //    TON_2 { ExternalWritable := 'False'} : TON;
   //    TON_3 { ExternalWritable := 'False'} : TON;
   //    TON_4 { ExternalWritable := 'False'} : TON;
   // END_VAR
BEGIN
END_DATA_BLOCK

DATA_BLOCK "n0061-uc22-el001-k30001_SN51_2"   // DB1121, F_DB
VERSION : 0.1
// stored: AutoNumber true, DBAccessibleFromOPCUA true, DBAccessibleFromWebserver true, InstanceOfName 00_Push-Button_Input, InstanceOfType FB
"00_Push-Button_Input"
   // VAR_INPUT
   //    IN_1 : Bool;
   //    IN_2 : Bool;
   //    IN_3 : Bool;
   //    IN_4 : Bool;
   //    ON_Tristate : Bool;
   //    ON_Lamp : Bool;
   //    Reset : Bool;
   //    REAC_DELAY { ExternalWritable := 'False'} : Time;
   //    Bypass_ET200 : Bool;
   // END_VAR
   // VAR_OUTPUT
   //    OUT_1 : Bool;
   //    OUT_2 : Bool;
   //    OUT_3 : Bool;
   //    OUT_4 : Bool;
   //    Diag_1 : Bool;
   //    Diag_2 : Bool;
   //    Diag_3 : Bool;
   //    Diag_4 : Bool;
   //    Lamp_1 : Bool;
   //    Lamp_2 : Bool;
   //    Lamp_3 : Bool;
   //    Lamp_4 : Bool;
   // END_VAR
   // VAR
   //    ESTOP_1 { S7_SetPoint := 'True'} : ESTOP1;
   //    ESTOP_2 { S7_SetPoint := 'True'} : ESTOP1;
   //    ESTOP_3 { S7_SetPoint := 'True'} : ESTOP1;
   //    ESTOP_4 { S7_SetPoint := 'True'} : ESTOP1;
   //    TON_1 { ExternalWritable := 'False'} : TON;
   //    TON_2 { ExternalWritable := 'False'} : TON;
   //    TON_3 { ExternalWritable := 'False'} : TON;
   //    TON_4 { ExternalWritable := 'False'} : TON;
   // END_VAR
BEGIN
END_DATA_BLOCK

DATA_BLOCK "n0061-uc22-el001-k30001_SN51_3"   // DB1122, F_DB
VERSION : 0.1
// stored: AutoNumber true, DBAccessibleFromOPCUA true, DBAccessibleFromWebserver true, InstanceOfName 00_Push-Button_Input, InstanceOfType FB
"00_Push-Button_Input"
   // VAR_INPUT
   //    IN_1 : Bool;
   //    IN_2 : Bool;
   //    IN_3 : Bool;
   //    IN_4 : Bool;
   //    ON_Tristate : Bool;
   //    ON_Lamp : Bool;
   //    Reset : Bool;
   //    REAC_DELAY { ExternalWritable := 'False'} : Time;
   //    Bypass_ET200 : Bool;
   // END_VAR
   // VAR_OUTPUT
   //    OUT_1 : Bool;
   //    OUT_2 : Bool;
   //    OUT_3 : Bool;
   //    OUT_4 : Bool;
   //    Diag_1 : Bool;
   //    Diag_2 : Bool;
   //    Diag_3 : Bool;
   //    Diag_4 : Bool;
   //    Lamp_1 : Bool;
   //    Lamp_2 : Bool;
   //    Lamp_3 : Bool;
   //    Lamp_4 : Bool;
   // END_VAR
   // VAR
   //    ESTOP_1 { S7_SetPoint := 'True'} : ESTOP1;
   //    ESTOP_2 { S7_SetPoint := 'True'} : ESTOP1;
   //    ESTOP_3 { S7_SetPoint := 'True'} : ESTOP1;
   //    ESTOP_4 { S7_SetPoint := 'True'} : ESTOP1;
   //    TON_1 { ExternalWritable := 'False'} : TON;
   //    TON_2 { ExternalWritable := 'False'} : TON;
   //    TON_3 { ExternalWritable := 'False'} : TON;
   //    TON_4 { ExternalWritable := 'False'} : TON;
   // END_VAR
BEGIN
END_DATA_BLOCK

DATA_BLOCK "n0061-uc22-el001-k30001_SN51_4"   // DB1123, F_DB
VERSION : 0.1
// stored: AutoNumber true, DBAccessibleFromOPCUA true, DBAccessibleFromWebserver true, InstanceOfName 00_Push-Button_Input, InstanceOfType FB
"00_Push-Button_Input"
   // VAR_INPUT
   //    IN_1 : Bool;
   //    IN_2 : Bool;
   //    IN_3 : Bool;
   //    IN_4 : Bool;
   //    ON_Tristate : Bool;
   //    ON_Lamp : Bool;
   //    Reset : Bool;
   //    REAC_DELAY { ExternalWritable := 'False'} : Time;
   //    Bypass_ET200 : Bool;
   // END_VAR
   // VAR_OUTPUT
   //    OUT_1 : Bool;
   //    OUT_2 : Bool;
   //    OUT_3 : Bool;
   //    OUT_4 : Bool;
   //    Diag_1 : Bool;
   //    Diag_2 : Bool;
   //    Diag_3 : Bool;
   //    Diag_4 : Bool;
   //    Lamp_1 : Bool;
   //    Lamp_2 : Bool;
   //    Lamp_3 : Bool;
   //    Lamp_4 : Bool;
   // END_VAR
   // VAR
   //    ESTOP_1 { S7_SetPoint := 'True'} : ESTOP1;
   //    ESTOP_2 { S7_SetPoint := 'True'} : ESTOP1;
   //    ESTOP_3 { S7_SetPoint := 'True'} : ESTOP1;
   //    ESTOP_4 { S7_SetPoint := 'True'} : ESTOP1;
   //    TON_1 { ExternalWritable := 'False'} : TON;
   //    TON_2 { ExternalWritable := 'False'} : TON;
   //    TON_3 { ExternalWritable := 'False'} : TON;
   //    TON_4 { ExternalWritable := 'False'} : TON;
   // END_VAR
BEGIN
END_DATA_BLOCK

DATA_BLOCK "n0057-uc224-xn10_SN51_1"   // DB1124, F_DB
VERSION : 0.1
// stored: AutoNumber true, DBAccessibleFromOPCUA true, DBAccessibleFromWebserver true, InstanceOfName 00_Push-Button_Input, InstanceOfType FB
"00_Push-Button_Input"
   // VAR_INPUT
   //    IN_1 : Bool;
   //    IN_2 : Bool;
   //    IN_3 : Bool;
   //    IN_4 : Bool;
   //    ON_Tristate : Bool;
   //    ON_Lamp : Bool;
   //    Reset : Bool;
   //    REAC_DELAY { ExternalWritable := 'False'} : Time;
   //    Bypass_ET200 : Bool;
   // END_VAR
   // VAR_OUTPUT
   //    OUT_1 : Bool;
   //    OUT_2 : Bool;
   //    OUT_3 : Bool;
   //    OUT_4 : Bool;
   //    Diag_1 : Bool;
   //    Diag_2 : Bool;
   //    Diag_3 : Bool;
   //    Diag_4 : Bool;
   //    Lamp_1 : Bool;
   //    Lamp_2 : Bool;
   //    Lamp_3 : Bool;
   //    Lamp_4 : Bool;
   // END_VAR
   // VAR
   //    ESTOP_1 { S7_SetPoint := 'True'} : ESTOP1;
   //    ESTOP_2 { S7_SetPoint := 'True'} : ESTOP1;
   //    ESTOP_3 { S7_SetPoint := 'True'} : ESTOP1;
   //    ESTOP_4 { S7_SetPoint := 'True'} : ESTOP1;
   //    TON_1 { ExternalWritable := 'False'} : TON;
   //    TON_2 { ExternalWritable := 'False'} : TON;
   //    TON_3 { ExternalWritable := 'False'} : TON;
   //    TON_4 { ExternalWritable := 'False'} : TON;
   // END_VAR
BEGIN
END_DATA_BLOCK

DATA_BLOCK "n0057-uc224-xn10_SN51_2"   // DB1125, F_DB
VERSION : 0.1
// stored: AutoNumber true, DBAccessibleFromOPCUA true, DBAccessibleFromWebserver true, InstanceOfName 00_Push-Button_Input, InstanceOfType FB
"00_Push-Button_Input"
   // VAR_INPUT
   //    IN_1 : Bool;
   //    IN_2 : Bool;
   //    IN_3 : Bool;
   //    IN_4 : Bool;
   //    ON_Tristate : Bool;
   //    ON_Lamp : Bool;
   //    Reset : Bool;
   //    REAC_DELAY { ExternalWritable := 'False'} : Time;
   //    Bypass_ET200 : Bool;
   // END_VAR
   // VAR_OUTPUT
   //    OUT_1 : Bool;
   //    OUT_2 : Bool;
   //    OUT_3 : Bool;
   //    OUT_4 : Bool;
   //    Diag_1 : Bool;
   //    Diag_2 : Bool;
   //    Diag_3 : Bool;
   //    Diag_4 : Bool;
   //    Lamp_1 : Bool;
   //    Lamp_2 : Bool;
   //    Lamp_3 : Bool;
   //    Lamp_4 : Bool;
   // END_VAR
   // VAR
   //    ESTOP_1 { S7_SetPoint := 'True'} : ESTOP1;
   //    ESTOP_2 { S7_SetPoint := 'True'} : ESTOP1;
   //    ESTOP_3 { S7_SetPoint := 'True'} : ESTOP1;
   //    ESTOP_4 { S7_SetPoint := 'True'} : ESTOP1;
   //    TON_1 { ExternalWritable := 'False'} : TON;
   //    TON_2 { ExternalWritable := 'False'} : TON;
   //    TON_3 { ExternalWritable := 'False'} : TON;
   //    TON_4 { ExternalWritable := 'False'} : TON;
   // END_VAR
BEGIN
END_DATA_BLOCK

DATA_BLOCK "n0066-uc21-el001-k30001_SN51_1"   // DB1126, F_DB
VERSION : 0.1
// stored: AutoNumber true, DBAccessibleFromOPCUA true, DBAccessibleFromWebserver true, InstanceOfName 00_Push-Button_Input, InstanceOfType FB
"00_Push-Button_Input"
   // VAR_INPUT
   //    IN_1 : Bool;
   //    IN_2 : Bool;
   //    IN_3 : Bool;
   //    IN_4 : Bool;
   //    ON_Tristate : Bool;
   //    ON_Lamp : Bool;
   //    Reset : Bool;
   //    REAC_DELAY { ExternalWritable := 'False'} : Time;
   //    Bypass_ET200 : Bool;
   // END_VAR
   // VAR_OUTPUT
   //    OUT_1 : Bool;
   //    OUT_2 : Bool;
   //    OUT_3 : Bool;
   //    OUT_4 : Bool;
   //    Diag_1 : Bool;
   //    Diag_2 : Bool;
   //    Diag_3 : Bool;
   //    Diag_4 : Bool;
   //    Lamp_1 : Bool;
   //    Lamp_2 : Bool;
   //    Lamp_3 : Bool;
   //    Lamp_4 : Bool;
   // END_VAR
   // VAR
   //    ESTOP_1 { S7_SetPoint := 'True'} : ESTOP1;
   //    ESTOP_2 { S7_SetPoint := 'True'} : ESTOP1;
   //    ESTOP_3 { S7_SetPoint := 'True'} : ESTOP1;
   //    ESTOP_4 { S7_SetPoint := 'True'} : ESTOP1;
   //    TON_1 { ExternalWritable := 'False'} : TON;
   //    TON_2 { ExternalWritable := 'False'} : TON;
   //    TON_3 { ExternalWritable := 'False'} : TON;
   //    TON_4 { ExternalWritable := 'False'} : TON;
   // END_VAR
BEGIN
END_DATA_BLOCK

DATA_BLOCK "n0066-uc21-el001-k30001_SN51_2"   // DB1127, F_DB
VERSION : 0.1
// stored: AutoNumber true, DBAccessibleFromOPCUA true, DBAccessibleFromWebserver true, InstanceOfName 00_Push-Button_Input, InstanceOfType FB
"00_Push-Button_Input"
   // VAR_INPUT
   //    IN_1 : Bool;
   //    IN_2 : Bool;
   //    IN_3 : Bool;
   //    IN_4 : Bool;
   //    ON_Tristate : Bool;
   //    ON_Lamp : Bool;
   //    Reset : Bool;
   //    REAC_DELAY { ExternalWritable := 'False'} : Time;
   //    Bypass_ET200 : Bool;
   // END_VAR
   // VAR_OUTPUT
   //    OUT_1 : Bool;
   //    OUT_2 : Bool;
   //    OUT_3 : Bool;
   //    OUT_4 : Bool;
   //    Diag_1 : Bool;
   //    Diag_2 : Bool;
   //    Diag_3 : Bool;
   //    Diag_4 : Bool;
   //    Lamp_1 : Bool;
   //    Lamp_2 : Bool;
   //    Lamp_3 : Bool;
   //    Lamp_4 : Bool;
   // END_VAR
   // VAR
   //    ESTOP_1 { S7_SetPoint := 'True'} : ESTOP1;
   //    ESTOP_2 { S7_SetPoint := 'True'} : ESTOP1;
   //    ESTOP_3 { S7_SetPoint := 'True'} : ESTOP1;
   //    ESTOP_4 { S7_SetPoint := 'True'} : ESTOP1;
   //    TON_1 { ExternalWritable := 'False'} : TON;
   //    TON_2 { ExternalWritable := 'False'} : TON;
   //    TON_3 { ExternalWritable := 'False'} : TON;
   //    TON_4 { ExternalWritable := 'False'} : TON;
   // END_VAR
BEGIN
END_DATA_BLOCK

DATA_BLOCK "n0066-uc21-el001-k30001_SN51_3"   // DB1128, F_DB
VERSION : 0.1
// stored: AutoNumber true, DBAccessibleFromOPCUA true, DBAccessibleFromWebserver true, InstanceOfName 00_Push-Button_Input, InstanceOfType FB
"00_Push-Button_Input"
   // VAR_INPUT
   //    IN_1 : Bool;
   //    IN_2 : Bool;
   //    IN_3 : Bool;
   //    IN_4 : Bool;
   //    ON_Tristate : Bool;
   //    ON_Lamp : Bool;
   //    Reset : Bool;
   //    REAC_DELAY { ExternalWritable := 'False'} : Time;
   //    Bypass_ET200 : Bool;
   // END_VAR
   // VAR_OUTPUT
   //    OUT_1 : Bool;
   //    OUT_2 : Bool;
   //    OUT_3 : Bool;
   //    OUT_4 : Bool;
   //    Diag_1 : Bool;
   //    Diag_2 : Bool;
   //    Diag_3 : Bool;
   //    Diag_4 : Bool;
   //    Lamp_1 : Bool;
   //    Lamp_2 : Bool;
   //    Lamp_3 : Bool;
   //    Lamp_4 : Bool;
   // END_VAR
   // VAR
   //    ESTOP_1 { S7_SetPoint := 'True'} : ESTOP1;
   //    ESTOP_2 { S7_SetPoint := 'True'} : ESTOP1;
   //    ESTOP_3 { S7_SetPoint := 'True'} : ESTOP1;
   //    ESTOP_4 { S7_SetPoint := 'True'} : ESTOP1;
   //    TON_1 { ExternalWritable := 'False'} : TON;
   //    TON_2 { ExternalWritable := 'False'} : TON;
   //    TON_3 { ExternalWritable := 'False'} : TON;
   //    TON_4 { ExternalWritable := 'False'} : TON;
   // END_VAR
BEGIN
END_DATA_BLOCK

DATA_BLOCK "n0067-uc214-xn10_SN51_1"   // DB1129, F_DB
VERSION : 0.1
// stored: AutoNumber true, DBAccessibleFromOPCUA true, DBAccessibleFromWebserver true, InstanceOfName 00_Push-Button_Input, InstanceOfType FB
"00_Push-Button_Input"
   // VAR_INPUT
   //    IN_1 : Bool;
   //    IN_2 : Bool;
   //    IN_3 : Bool;
   //    IN_4 : Bool;
   //    ON_Tristate : Bool;
   //    ON_Lamp : Bool;
   //    Reset : Bool;
   //    REAC_DELAY { ExternalWritable := 'False'} : Time;
   //    Bypass_ET200 : Bool;
   // END_VAR
   // VAR_OUTPUT
   //    OUT_1 : Bool;
   //    OUT_2 : Bool;
   //    OUT_3 : Bool;
   //    OUT_4 : Bool;
   //    Diag_1 : Bool;
   //    Diag_2 : Bool;
   //    Diag_3 : Bool;
   //    Diag_4 : Bool;
   //    Lamp_1 : Bool;
   //    Lamp_2 : Bool;
   //    Lamp_3 : Bool;
   //    Lamp_4 : Bool;
   // END_VAR
   // VAR
   //    ESTOP_1 { S7_SetPoint := 'True'} : ESTOP1;
   //    ESTOP_2 { S7_SetPoint := 'True'} : ESTOP1;
   //    ESTOP_3 { S7_SetPoint := 'True'} : ESTOP1;
   //    ESTOP_4 { S7_SetPoint := 'True'} : ESTOP1;
   //    TON_1 { ExternalWritable := 'False'} : TON;
   //    TON_2 { ExternalWritable := 'False'} : TON;
   //    TON_3 { ExternalWritable := 'False'} : TON;
   //    TON_4 { ExternalWritable := 'False'} : TON;
   // END_VAR
BEGIN
END_DATA_BLOCK

DATA_BLOCK "n0067-uc214-xn10_SN51_2"   // DB1130, F_DB
VERSION : 0.1
// stored: AutoNumber true, DBAccessibleFromOPCUA true, DBAccessibleFromWebserver true, InstanceOfName 00_Push-Button_Input, InstanceOfType FB
"00_Push-Button_Input"
   // VAR_INPUT
   //    IN_1 : Bool;
   //    IN_2 : Bool;
   //    IN_3 : Bool;
   //    IN_4 : Bool;
   //    ON_Tristate : Bool;
   //    ON_Lamp : Bool;
   //    Reset : Bool;
   //    REAC_DELAY { ExternalWritable := 'False'} : Time;
   //    Bypass_ET200 : Bool;
   // END_VAR
   // VAR_OUTPUT
   //    OUT_1 : Bool;
   //    OUT_2 : Bool;
   //    OUT_3 : Bool;
   //    OUT_4 : Bool;
   //    Diag_1 : Bool;
   //    Diag_2 : Bool;
   //    Diag_3 : Bool;
   //    Diag_4 : Bool;
   //    Lamp_1 : Bool;
   //    Lamp_2 : Bool;
   //    Lamp_3 : Bool;
   //    Lamp_4 : Bool;
   // END_VAR
   // VAR
   //    ESTOP_1 { S7_SetPoint := 'True'} : ESTOP1;
   //    ESTOP_2 { S7_SetPoint := 'True'} : ESTOP1;
   //    ESTOP_3 { S7_SetPoint := 'True'} : ESTOP1;
   //    ESTOP_4 { S7_SetPoint := 'True'} : ESTOP1;
   //    TON_1 { ExternalWritable := 'False'} : TON;
   //    TON_2 { ExternalWritable := 'False'} : TON;
   //    TON_3 { ExternalWritable := 'False'} : TON;
   //    TON_4 { ExternalWritable := 'False'} : TON;
   // END_VAR
BEGIN
END_DATA_BLOCK

DATA_BLOCK "n0070-uf31-el001-k30001_SN51_1"   // DB1131, F_DB
VERSION : 0.1
// stored: AutoNumber true, DBAccessibleFromOPCUA true, DBAccessibleFromWebserver true, InstanceOfName 00_Push-Button_Input, InstanceOfType FB
"00_Push-Button_Input"
   // VAR_INPUT
   //    IN_1 : Bool;
   //    IN_2 : Bool;
   //    IN_3 : Bool;
   //    IN_4 : Bool;
   //    ON_Tristate : Bool;
   //    ON_Lamp : Bool;
   //    Reset : Bool;
   //    REAC_DELAY { ExternalWritable := 'False'} : Time;
   //    Bypass_ET200 : Bool;
   // END_VAR
   // VAR_OUTPUT
   //    OUT_1 : Bool;
   //    OUT_2 : Bool;
   //    OUT_3 : Bool;
   //    OUT_4 : Bool;
   //    Diag_1 : Bool;
   //    Diag_2 : Bool;
   //    Diag_3 : Bool;
   //    Diag_4 : Bool;
   //    Lamp_1 : Bool;
   //    Lamp_2 : Bool;
   //    Lamp_3 : Bool;
   //    Lamp_4 : Bool;
   // END_VAR
   // VAR
   //    ESTOP_1 { S7_SetPoint := 'True'} : ESTOP1;
   //    ESTOP_2 { S7_SetPoint := 'True'} : ESTOP1;
   //    ESTOP_3 { S7_SetPoint := 'True'} : ESTOP1;
   //    ESTOP_4 { S7_SetPoint := 'True'} : ESTOP1;
   //    TON_1 { ExternalWritable := 'False'} : TON;
   //    TON_2 { ExternalWritable := 'False'} : TON;
   //    TON_3 { ExternalWritable := 'False'} : TON;
   //    TON_4 { ExternalWritable := 'False'} : TON;
   // END_VAR
BEGIN
END_DATA_BLOCK

DATA_BLOCK "n0072-uf51-el001-k30001_SN51_1"   // DB1132, F_DB
VERSION : 0.1
// stored: AutoNumber true, DBAccessibleFromOPCUA true, DBAccessibleFromWebserver true, InstanceOfName 00_Push-Button_Input, InstanceOfType FB
"00_Push-Button_Input"
   // VAR_INPUT
   //    IN_1 : Bool;
   //    IN_2 : Bool;
   //    IN_3 : Bool;
   //    IN_4 : Bool;
   //    ON_Tristate : Bool;
   //    ON_Lamp : Bool;
   //    Reset : Bool;
   //    REAC_DELAY { ExternalWritable := 'False'} : Time;
   //    Bypass_ET200 : Bool;
   // END_VAR
   // VAR_OUTPUT
   //    OUT_1 : Bool;
   //    OUT_2 : Bool;
   //    OUT_3 : Bool;
   //    OUT_4 : Bool;
   //    Diag_1 : Bool;
   //    Diag_2 : Bool;
   //    Diag_3 : Bool;
   //    Diag_4 : Bool;
   //    Lamp_1 : Bool;
   //    Lamp_2 : Bool;
   //    Lamp_3 : Bool;
   //    Lamp_4 : Bool;
   // END_VAR
   // VAR
   //    ESTOP_1 { S7_SetPoint := 'True'} : ESTOP1;
   //    ESTOP_2 { S7_SetPoint := 'True'} : ESTOP1;
   //    ESTOP_3 { S7_SetPoint := 'True'} : ESTOP1;
   //    ESTOP_4 { S7_SetPoint := 'True'} : ESTOP1;
   //    TON_1 { ExternalWritable := 'False'} : TON;
   //    TON_2 { ExternalWritable := 'False'} : TON;
   //    TON_3 { ExternalWritable := 'False'} : TON;
   //    TON_4 { ExternalWritable := 'False'} : TON;
   // END_VAR
BEGIN
END_DATA_BLOCK

DATA_BLOCK "n0080-uf511-xn10_SN51_1"   // DB1133, F_DB
VERSION : 0.1
// stored: AutoNumber true, DBAccessibleFromOPCUA true, DBAccessibleFromWebserver true, InstanceOfName 00_Push-Button_Input, InstanceOfType FB
"00_Push-Button_Input"
   // VAR_INPUT
   //    IN_1 : Bool;
   //    IN_2 : Bool;
   //    IN_3 : Bool;
   //    IN_4 : Bool;
   //    ON_Tristate : Bool;
   //    ON_Lamp : Bool;
   //    Reset : Bool;
   //    REAC_DELAY { ExternalWritable := 'False'} : Time;
   //    Bypass_ET200 : Bool;
   // END_VAR
   // VAR_OUTPUT
   //    OUT_1 : Bool;
   //    OUT_2 : Bool;
   //    OUT_3 : Bool;
   //    OUT_4 : Bool;
   //    Diag_1 : Bool;
   //    Diag_2 : Bool;
   //    Diag_3 : Bool;
   //    Diag_4 : Bool;
   //    Lamp_1 : Bool;
   //    Lamp_2 : Bool;
   //    Lamp_3 : Bool;
   //    Lamp_4 : Bool;
   // END_VAR
   // VAR
   //    ESTOP_1 { S7_SetPoint := 'True'} : ESTOP1;
   //    ESTOP_2 { S7_SetPoint := 'True'} : ESTOP1;
   //    ESTOP_3 { S7_SetPoint := 'True'} : ESTOP1;
   //    ESTOP_4 { S7_SetPoint := 'True'} : ESTOP1;
   //    TON_1 { ExternalWritable := 'False'} : TON;
   //    TON_2 { ExternalWritable := 'False'} : TON;
   //    TON_3 { ExternalWritable := 'False'} : TON;
   //    TON_4 { ExternalWritable := 'False'} : TON;
   // END_VAR
BEGIN
END_DATA_BLOCK

DATA_BLOCK "n0073-ifg31-el001-k30001_SN51_1"   // DB1134, F_DB
VERSION : 0.1
// stored: AutoNumber true, DBAccessibleFromOPCUA true, DBAccessibleFromWebserver true, InstanceOfName 00_Push-Button_Input, InstanceOfType FB
"00_Push-Button_Input"
   // VAR_INPUT
   //    IN_1 : Bool;
   //    IN_2 : Bool;
   //    IN_3 : Bool;
   //    IN_4 : Bool;
   //    ON_Tristate : Bool;
   //    ON_Lamp : Bool;
   //    Reset : Bool;
   //    REAC_DELAY { ExternalWritable := 'False'} : Time;
   //    Bypass_ET200 : Bool;
   // END_VAR
   // VAR_OUTPUT
   //    OUT_1 : Bool;
   //    OUT_2 : Bool;
   //    OUT_3 : Bool;
   //    OUT_4 : Bool;
   //    Diag_1 : Bool;
   //    Diag_2 : Bool;
   //    Diag_3 : Bool;
   //    Diag_4 : Bool;
   //    Lamp_1 : Bool;
   //    Lamp_2 : Bool;
   //    Lamp_3 : Bool;
   //    Lamp_4 : Bool;
   // END_VAR
   // VAR
   //    ESTOP_1 { S7_SetPoint := 'True'} : ESTOP1;
   //    ESTOP_2 { S7_SetPoint := 'True'} : ESTOP1;
   //    ESTOP_3 { S7_SetPoint := 'True'} : ESTOP1;
   //    ESTOP_4 { S7_SetPoint := 'True'} : ESTOP1;
   //    TON_1 { ExternalWritable := 'False'} : TON;
   //    TON_2 { ExternalWritable := 'False'} : TON;
   //    TON_3 { ExternalWritable := 'False'} : TON;
   //    TON_4 { ExternalWritable := 'False'} : TON;
   // END_VAR
BEGIN
END_DATA_BLOCK

DATA_BLOCK "n0073-ifg31-el001-k30001_SN51_2"   // DB1135, F_DB
VERSION : 0.1
// stored: AutoNumber true, DBAccessibleFromOPCUA true, DBAccessibleFromWebserver true, InstanceOfName 00_Push-Button_Input, InstanceOfType FB
"00_Push-Button_Input"
   // VAR_INPUT
   //    IN_1 : Bool;
   //    IN_2 : Bool;
   //    IN_3 : Bool;
   //    IN_4 : Bool;
   //    ON_Tristate : Bool;
   //    ON_Lamp : Bool;
   //    Reset : Bool;
   //    REAC_DELAY { ExternalWritable := 'False'} : Time;
   //    Bypass_ET200 : Bool;
   // END_VAR
   // VAR_OUTPUT
   //    OUT_1 : Bool;
   //    OUT_2 : Bool;
   //    OUT_3 : Bool;
   //    OUT_4 : Bool;
   //    Diag_1 : Bool;
   //    Diag_2 : Bool;
   //    Diag_3 : Bool;
   //    Diag_4 : Bool;
   //    Lamp_1 : Bool;
   //    Lamp_2 : Bool;
   //    Lamp_3 : Bool;
   //    Lamp_4 : Bool;
   // END_VAR
   // VAR
   //    ESTOP_1 { S7_SetPoint := 'True'} : ESTOP1;
   //    ESTOP_2 { S7_SetPoint := 'True'} : ESTOP1;
   //    ESTOP_3 { S7_SetPoint := 'True'} : ESTOP1;
   //    ESTOP_4 { S7_SetPoint := 'True'} : ESTOP1;
   //    TON_1 { ExternalWritable := 'False'} : TON;
   //    TON_2 { ExternalWritable := 'False'} : TON;
   //    TON_3 { ExternalWritable := 'False'} : TON;
   //    TON_4 { ExternalWritable := 'False'} : TON;
   // END_VAR
BEGIN
END_DATA_BLOCK

DATA_BLOCK "n0074-ifg41-el001-k30001_SN51_1"   // DB1136, F_DB
VERSION : 0.1
// stored: AutoNumber true, DBAccessibleFromOPCUA true, DBAccessibleFromWebserver true, InstanceOfName 00_Push-Button_Input, InstanceOfType FB
"00_Push-Button_Input"
   // VAR_INPUT
   //    IN_1 : Bool;
   //    IN_2 : Bool;
   //    IN_3 : Bool;
   //    IN_4 : Bool;
   //    ON_Tristate : Bool;
   //    ON_Lamp : Bool;
   //    Reset : Bool;
   //    REAC_DELAY { ExternalWritable := 'False'} : Time;
   //    Bypass_ET200 : Bool;
   // END_VAR
   // VAR_OUTPUT
   //    OUT_1 : Bool;
   //    OUT_2 : Bool;
   //    OUT_3 : Bool;
   //    OUT_4 : Bool;
   //    Diag_1 : Bool;
   //    Diag_2 : Bool;
   //    Diag_3 : Bool;
   //    Diag_4 : Bool;
   //    Lamp_1 : Bool;
   //    Lamp_2 : Bool;
   //    Lamp_3 : Bool;
   //    Lamp_4 : Bool;
   // END_VAR
   // VAR
   //    ESTOP_1 { S7_SetPoint := 'True'} : ESTOP1;
   //    ESTOP_2 { S7_SetPoint := 'True'} : ESTOP1;
   //    ESTOP_3 { S7_SetPoint := 'True'} : ESTOP1;
   //    ESTOP_4 { S7_SetPoint := 'True'} : ESTOP1;
   //    TON_1 { ExternalWritable := 'False'} : TON;
   //    TON_2 { ExternalWritable := 'False'} : TON;
   //    TON_3 { ExternalWritable := 'False'} : TON;
   //    TON_4 { ExternalWritable := 'False'} : TON;
   // END_VAR
BEGIN
END_DATA_BLOCK

DATA_BLOCK "n0075-uf32-el001-k30001_SN51_1"   // DB1137, F_DB
VERSION : 0.1
// stored: AutoNumber true, DBAccessibleFromOPCUA true, DBAccessibleFromWebserver true, InstanceOfName 00_Push-Button_Input, InstanceOfType FB
"00_Push-Button_Input"
   // VAR_INPUT
   //    IN_1 : Bool;
   //    IN_2 : Bool;
   //    IN_3 : Bool;
   //    IN_4 : Bool;
   //    ON_Tristate : Bool;
   //    ON_Lamp : Bool;
   //    Reset : Bool;
   //    REAC_DELAY { ExternalWritable := 'False'} : Time;
   //    Bypass_ET200 : Bool;
   // END_VAR
   // VAR_OUTPUT
   //    OUT_1 : Bool;
   //    OUT_2 : Bool;
   //    OUT_3 : Bool;
   //    OUT_4 : Bool;
   //    Diag_1 : Bool;
   //    Diag_2 : Bool;
   //    Diag_3 : Bool;
   //    Diag_4 : Bool;
   //    Lamp_1 : Bool;
   //    Lamp_2 : Bool;
   //    Lamp_3 : Bool;
   //    Lamp_4 : Bool;
   // END_VAR
   // VAR
   //    ESTOP_1 { S7_SetPoint := 'True'} : ESTOP1;
   //    ESTOP_2 { S7_SetPoint := 'True'} : ESTOP1;
   //    ESTOP_3 { S7_SetPoint := 'True'} : ESTOP1;
   //    ESTOP_4 { S7_SetPoint := 'True'} : ESTOP1;
   //    TON_1 { ExternalWritable := 'False'} : TON;
   //    TON_2 { ExternalWritable := 'False'} : TON;
   //    TON_3 { ExternalWritable := 'False'} : TON;
   //    TON_4 { ExternalWritable := 'False'} : TON;
   // END_VAR
BEGIN
END_DATA_BLOCK

DATA_BLOCK "n0082-zp002-el001-k30001_SN51_1"   // DB1138, F_DB
VERSION : 0.1
// stored: AutoNumber true, DBAccessibleFromOPCUA true, DBAccessibleFromWebserver true, InstanceOfName 00_Push-Button_Input, InstanceOfType FB
"00_Push-Button_Input"
   // VAR_INPUT
   //    IN_1 : Bool;
   //    IN_2 : Bool;
   //    IN_3 : Bool;
   //    IN_4 : Bool;
   //    ON_Tristate : Bool;
   //    ON_Lamp : Bool;
   //    Reset : Bool;
   //    REAC_DELAY { ExternalWritable := 'False'} : Time;
   //    Bypass_ET200 : Bool;
   // END_VAR
   // VAR_OUTPUT
   //    OUT_1 : Bool;
   //    OUT_2 : Bool;
   //    OUT_3 : Bool;
   //    OUT_4 : Bool;
   //    Diag_1 : Bool;
   //    Diag_2 : Bool;
   //    Diag_3 : Bool;
   //    Diag_4 : Bool;
   //    Lamp_1 : Bool;
   //    Lamp_2 : Bool;
   //    Lamp_3 : Bool;
   //    Lamp_4 : Bool;
   // END_VAR
   // VAR
   //    ESTOP_1 { S7_SetPoint := 'True'} : ESTOP1;
   //    ESTOP_2 { S7_SetPoint := 'True'} : ESTOP1;
   //    ESTOP_3 { S7_SetPoint := 'True'} : ESTOP1;
   //    ESTOP_4 { S7_SetPoint := 'True'} : ESTOP1;
   //    TON_1 { ExternalWritable := 'False'} : TON;
   //    TON_2 { ExternalWritable := 'False'} : TON;
   //    TON_3 { ExternalWritable := 'False'} : TON;
   //    TON_4 { ExternalWritable := 'False'} : TON;
   // END_VAR
BEGIN
END_DATA_BLOCK

DATA_BLOCK "n0083-lv001-el001-k30001_SN51_1"   // DB1139, F_DB
VERSION : 0.1
// stored: AutoNumber true, DBAccessibleFromOPCUA true, DBAccessibleFromWebserver true, InstanceOfName 00_Push-Button_Input, InstanceOfType FB
"00_Push-Button_Input"
   // VAR_INPUT
   //    IN_1 : Bool;
   //    IN_2 : Bool;
   //    IN_3 : Bool;
   //    IN_4 : Bool;
   //    ON_Tristate : Bool;
   //    ON_Lamp : Bool;
   //    Reset : Bool;
   //    REAC_DELAY { ExternalWritable := 'False'} : Time;
   //    Bypass_ET200 : Bool;
   // END_VAR
   // VAR_OUTPUT
   //    OUT_1 : Bool;
   //    OUT_2 : Bool;
   //    OUT_3 : Bool;
   //    OUT_4 : Bool;
   //    Diag_1 : Bool;
   //    Diag_2 : Bool;
   //    Diag_3 : Bool;
   //    Diag_4 : Bool;
   //    Lamp_1 : Bool;
   //    Lamp_2 : Bool;
   //    Lamp_3 : Bool;
   //    Lamp_4 : Bool;
   // END_VAR
   // VAR
   //    ESTOP_1 { S7_SetPoint := 'True'} : ESTOP1;
   //    ESTOP_2 { S7_SetPoint := 'True'} : ESTOP1;
   //    ESTOP_3 { S7_SetPoint := 'True'} : ESTOP1;
   //    ESTOP_4 { S7_SetPoint := 'True'} : ESTOP1;
   //    TON_1 { ExternalWritable := 'False'} : TON;
   //    TON_2 { ExternalWritable := 'False'} : TON;
   //    TON_3 { ExternalWritable := 'False'} : TON;
   //    TON_4 { ExternalWritable := 'False'} : TON;
   // END_VAR
BEGIN
END_DATA_BLOCK

DATA_BLOCK "n0084-lv001-el001-k30001_SN51_1"   // DB1140, F_DB
VERSION : 0.1
// stored: AutoNumber true, DBAccessibleFromOPCUA true, DBAccessibleFromWebserver true, InstanceOfName 00_Push-Button_Input, InstanceOfType FB
"00_Push-Button_Input"
   // VAR_INPUT
   //    IN_1 : Bool;
   //    IN_2 : Bool;
   //    IN_3 : Bool;
   //    IN_4 : Bool;
   //    ON_Tristate : Bool;
   //    ON_Lamp : Bool;
   //    Reset : Bool;
   //    REAC_DELAY { ExternalWritable := 'False'} : Time;
   //    Bypass_ET200 : Bool;
   // END_VAR
   // VAR_OUTPUT
   //    OUT_1 : Bool;
   //    OUT_2 : Bool;
   //    OUT_3 : Bool;
   //    OUT_4 : Bool;
   //    Diag_1 : Bool;
   //    Diag_2 : Bool;
   //    Diag_3 : Bool;
   //    Diag_4 : Bool;
   //    Lamp_1 : Bool;
   //    Lamp_2 : Bool;
   //    Lamp_3 : Bool;
   //    Lamp_4 : Bool;
   // END_VAR
   // VAR
   //    ESTOP_1 { S7_SetPoint := 'True'} : ESTOP1;
   //    ESTOP_2 { S7_SetPoint := 'True'} : ESTOP1;
   //    ESTOP_3 { S7_SetPoint := 'True'} : ESTOP1;
   //    ESTOP_4 { S7_SetPoint := 'True'} : ESTOP1;
   //    TON_1 { ExternalWritable := 'False'} : TON;
   //    TON_2 { ExternalWritable := 'False'} : TON;
   //    TON_3 { ExternalWritable := 'False'} : TON;
   //    TON_4 { ExternalWritable := 'False'} : TON;
   // END_VAR
BEGIN
END_DATA_BLOCK

DATA_BLOCK "n0085-uc29-el001-k30001_SN51_1"   // DB1141, F_DB
VERSION : 0.1
// stored: AutoNumber true, DBAccessibleFromOPCUA true, DBAccessibleFromWebserver true, InstanceOfName 00_Push-Button_Input, InstanceOfType FB
"00_Push-Button_Input"
   // VAR_INPUT
   //    IN_1 : Bool;
   //    IN_2 : Bool;
   //    IN_3 : Bool;
   //    IN_4 : Bool;
   //    ON_Tristate : Bool;
   //    ON_Lamp : Bool;
   //    Reset : Bool;
   //    REAC_DELAY { ExternalWritable := 'False'} : Time;
   //    Bypass_ET200 : Bool;
   // END_VAR
   // VAR_OUTPUT
   //    OUT_1 : Bool;
   //    OUT_2 : Bool;
   //    OUT_3 : Bool;
   //    OUT_4 : Bool;
   //    Diag_1 : Bool;
   //    Diag_2 : Bool;
   //    Diag_3 : Bool;
   //    Diag_4 : Bool;
   //    Lamp_1 : Bool;
   //    Lamp_2 : Bool;
   //    Lamp_3 : Bool;
   //    Lamp_4 : Bool;
   // END_VAR
   // VAR
   //    ESTOP_1 { S7_SetPoint := 'True'} : ESTOP1;
   //    ESTOP_2 { S7_SetPoint := 'True'} : ESTOP1;
   //    ESTOP_3 { S7_SetPoint := 'True'} : ESTOP1;
   //    ESTOP_4 { S7_SetPoint := 'True'} : ESTOP1;
   //    TON_1 { ExternalWritable := 'False'} : TON;
   //    TON_2 { ExternalWritable := 'False'} : TON;
   //    TON_3 { ExternalWritable := 'False'} : TON;
   //    TON_4 { ExternalWritable := 'False'} : TON;
   // END_VAR
BEGIN
END_DATA_BLOCK

DATA_BLOCK "n0085-uc29-el001-k30001_SN51_2"   // DB1142, F_DB
VERSION : 0.1
// stored: AutoNumber true, DBAccessibleFromOPCUA true, DBAccessibleFromWebserver true, InstanceOfName 00_Push-Button_Input, InstanceOfType FB
"00_Push-Button_Input"
   // VAR_INPUT
   //    IN_1 : Bool;
   //    IN_2 : Bool;
   //    IN_3 : Bool;
   //    IN_4 : Bool;
   //    ON_Tristate : Bool;
   //    ON_Lamp : Bool;
   //    Reset : Bool;
   //    REAC_DELAY { ExternalWritable := 'False'} : Time;
   //    Bypass_ET200 : Bool;
   // END_VAR
   // VAR_OUTPUT
   //    OUT_1 : Bool;
   //    OUT_2 : Bool;
   //    OUT_3 : Bool;
   //    OUT_4 : Bool;
   //    Diag_1 : Bool;
   //    Diag_2 : Bool;
   //    Diag_3 : Bool;
   //    Diag_4 : Bool;
   //    Lamp_1 : Bool;
   //    Lamp_2 : Bool;
   //    Lamp_3 : Bool;
   //    Lamp_4 : Bool;
   // END_VAR
   // VAR
   //    ESTOP_1 { S7_SetPoint := 'True'} : ESTOP1;
   //    ESTOP_2 { S7_SetPoint := 'True'} : ESTOP1;
   //    ESTOP_3 { S7_SetPoint := 'True'} : ESTOP1;
   //    ESTOP_4 { S7_SetPoint := 'True'} : ESTOP1;
   //    TON_1 { ExternalWritable := 'False'} : TON;
   //    TON_2 { ExternalWritable := 'False'} : TON;
   //    TON_3 { ExternalWritable := 'False'} : TON;
   //    TON_4 { ExternalWritable := 'False'} : TON;
   // END_VAR
BEGIN
END_DATA_BLOCK

DATA_BLOCK "n0091-zp001-el001-k30001_SN51_1"   // DB1143, F_DB
VERSION : 0.1
// stored: AutoNumber true, DBAccessibleFromOPCUA true, DBAccessibleFromWebserver true, InstanceOfName 00_Push-Button_Input, InstanceOfType FB
"00_Push-Button_Input"
   // VAR_INPUT
   //    IN_1 : Bool;
   //    IN_2 : Bool;
   //    IN_3 : Bool;
   //    IN_4 : Bool;
   //    ON_Tristate : Bool;
   //    ON_Lamp : Bool;
   //    Reset : Bool;
   //    REAC_DELAY { ExternalWritable := 'False'} : Time;
   //    Bypass_ET200 : Bool;
   // END_VAR
   // VAR_OUTPUT
   //    OUT_1 : Bool;
   //    OUT_2 : Bool;
   //    OUT_3 : Bool;
   //    OUT_4 : Bool;
   //    Diag_1 : Bool;
   //    Diag_2 : Bool;
   //    Diag_3 : Bool;
   //    Diag_4 : Bool;
   //    Lamp_1 : Bool;
   //    Lamp_2 : Bool;
   //    Lamp_3 : Bool;
   //    Lamp_4 : Bool;
   // END_VAR
   // VAR
   //    ESTOP_1 { S7_SetPoint := 'True'} : ESTOP1;
   //    ESTOP_2 { S7_SetPoint := 'True'} : ESTOP1;
   //    ESTOP_3 { S7_SetPoint := 'True'} : ESTOP1;
   //    ESTOP_4 { S7_SetPoint := 'True'} : ESTOP1;
   //    TON_1 { ExternalWritable := 'False'} : TON;
   //    TON_2 { ExternalWritable := 'False'} : TON;
   //    TON_3 { ExternalWritable := 'False'} : TON;
   //    TON_4 { ExternalWritable := 'False'} : TON;
   // END_VAR
BEGIN
END_DATA_BLOCK

DATA_BLOCK "n0091-zp001-el001-k30001_SN51_2"   // DB1144, F_DB
VERSION : 0.1
// stored: AutoNumber true, DBAccessibleFromOPCUA true, DBAccessibleFromWebserver true, InstanceOfName 00_Push-Button_Input, InstanceOfType FB
"00_Push-Button_Input"
   // VAR_INPUT
   //    IN_1 : Bool;
   //    IN_2 : Bool;
   //    IN_3 : Bool;
   //    IN_4 : Bool;
   //    ON_Tristate : Bool;
   //    ON_Lamp : Bool;
   //    Reset : Bool;
   //    REAC_DELAY { ExternalWritable := 'False'} : Time;
   //    Bypass_ET200 : Bool;
   // END_VAR
   // VAR_OUTPUT
   //    OUT_1 : Bool;
   //    OUT_2 : Bool;
   //    OUT_3 : Bool;
   //    OUT_4 : Bool;
   //    Diag_1 : Bool;
   //    Diag_2 : Bool;
   //    Diag_3 : Bool;
   //    Diag_4 : Bool;
   //    Lamp_1 : Bool;
   //    Lamp_2 : Bool;
   //    Lamp_3 : Bool;
   //    Lamp_4 : Bool;
   // END_VAR
   // VAR
   //    ESTOP_1 { S7_SetPoint := 'True'} : ESTOP1;
   //    ESTOP_2 { S7_SetPoint := 'True'} : ESTOP1;
   //    ESTOP_3 { S7_SetPoint := 'True'} : ESTOP1;
   //    ESTOP_4 { S7_SetPoint := 'True'} : ESTOP1;
   //    TON_1 { ExternalWritable := 'False'} : TON;
   //    TON_2 { ExternalWritable := 'False'} : TON;
   //    TON_3 { ExternalWritable := 'False'} : TON;
   //    TON_4 { ExternalWritable := 'False'} : TON;
   // END_VAR
BEGIN
END_DATA_BLOCK

DATA_BLOCK "n0093-ug7-el001-k30001_SN51_1"   // DB1145, F_DB
VERSION : 0.1
// stored: AutoNumber true, DBAccessibleFromOPCUA true, DBAccessibleFromWebserver true, InstanceOfName 00_Push-Button_Input, InstanceOfType FB
"00_Push-Button_Input"
   // VAR_INPUT
   //    IN_1 : Bool;
   //    IN_2 : Bool;
   //    IN_3 : Bool;
   //    IN_4 : Bool;
   //    ON_Tristate : Bool;
   //    ON_Lamp : Bool;
   //    Reset : Bool;
   //    REAC_DELAY { ExternalWritable := 'False'} : Time;
   //    Bypass_ET200 : Bool;
   // END_VAR
   // VAR_OUTPUT
   //    OUT_1 : Bool;
   //    OUT_2 : Bool;
   //    OUT_3 : Bool;
   //    OUT_4 : Bool;
   //    Diag_1 : Bool;
   //    Diag_2 : Bool;
   //    Diag_3 : Bool;
   //    Diag_4 : Bool;
   //    Lamp_1 : Bool;
   //    Lamp_2 : Bool;
   //    Lamp_3 : Bool;
   //    Lamp_4 : Bool;
   // END_VAR
   // VAR
   //    ESTOP_1 { S7_SetPoint := 'True'} : ESTOP1;
   //    ESTOP_2 { S7_SetPoint := 'True'} : ESTOP1;
   //    ESTOP_3 { S7_SetPoint := 'True'} : ESTOP1;
   //    ESTOP_4 { S7_SetPoint := 'True'} : ESTOP1;
   //    TON_1 { ExternalWritable := 'False'} : TON;
   //    TON_2 { ExternalWritable := 'False'} : TON;
   //    TON_3 { ExternalWritable := 'False'} : TON;
   //    TON_4 { ExternalWritable := 'False'} : TON;
   // END_VAR
BEGIN
END_DATA_BLOCK

DATA_BLOCK "n0093-ug7-el001-k30001_SN51_2"   // DB1146, F_DB
VERSION : 0.1
// stored: AutoNumber true, DBAccessibleFromOPCUA true, DBAccessibleFromWebserver true, InstanceOfName 00_Push-Button_Input, InstanceOfType FB
"00_Push-Button_Input"
   // VAR_INPUT
   //    IN_1 : Bool;
   //    IN_2 : Bool;
   //    IN_3 : Bool;
   //    IN_4 : Bool;
   //    ON_Tristate : Bool;
   //    ON_Lamp : Bool;
   //    Reset : Bool;
   //    REAC_DELAY { ExternalWritable := 'False'} : Time;
   //    Bypass_ET200 : Bool;
   // END_VAR
   // VAR_OUTPUT
   //    OUT_1 : Bool;
   //    OUT_2 : Bool;
   //    OUT_3 : Bool;
   //    OUT_4 : Bool;
   //    Diag_1 : Bool;
   //    Diag_2 : Bool;
   //    Diag_3 : Bool;
   //    Diag_4 : Bool;
   //    Lamp_1 : Bool;
   //    Lamp_2 : Bool;
   //    Lamp_3 : Bool;
   //    Lamp_4 : Bool;
   // END_VAR
   // VAR
   //    ESTOP_1 { S7_SetPoint := 'True'} : ESTOP1;
   //    ESTOP_2 { S7_SetPoint := 'True'} : ESTOP1;
   //    ESTOP_3 { S7_SetPoint := 'True'} : ESTOP1;
   //    ESTOP_4 { S7_SetPoint := 'True'} : ESTOP1;
   //    TON_1 { ExternalWritable := 'False'} : TON;
   //    TON_2 { ExternalWritable := 'False'} : TON;
   //    TON_3 { ExternalWritable := 'False'} : TON;
   //    TON_4 { ExternalWritable := 'False'} : TON;
   // END_VAR
BEGIN
END_DATA_BLOCK

DATA_BLOCK "n0093-ug7-el001-k30001_SN51_3"   // DB1147, F_DB
VERSION : 0.1
// stored: AutoNumber true, DBAccessibleFromOPCUA true, DBAccessibleFromWebserver true, InstanceOfName 00_Push-Button_Input, InstanceOfType FB
"00_Push-Button_Input"
   // VAR_INPUT
   //    IN_1 : Bool;
   //    IN_2 : Bool;
   //    IN_3 : Bool;
   //    IN_4 : Bool;
   //    ON_Tristate : Bool;
   //    ON_Lamp : Bool;
   //    Reset : Bool;
   //    REAC_DELAY { ExternalWritable := 'False'} : Time;
   //    Bypass_ET200 : Bool;
   // END_VAR
   // VAR_OUTPUT
   //    OUT_1 : Bool;
   //    OUT_2 : Bool;
   //    OUT_3 : Bool;
   //    OUT_4 : Bool;
   //    Diag_1 : Bool;
   //    Diag_2 : Bool;
   //    Diag_3 : Bool;
   //    Diag_4 : Bool;
   //    Lamp_1 : Bool;
   //    Lamp_2 : Bool;
   //    Lamp_3 : Bool;
   //    Lamp_4 : Bool;
   // END_VAR
   // VAR
   //    ESTOP_1 { S7_SetPoint := 'True'} : ESTOP1;
   //    ESTOP_2 { S7_SetPoint := 'True'} : ESTOP1;
   //    ESTOP_3 { S7_SetPoint := 'True'} : ESTOP1;
   //    ESTOP_4 { S7_SetPoint := 'True'} : ESTOP1;
   //    TON_1 { ExternalWritable := 'False'} : TON;
   //    TON_2 { ExternalWritable := 'False'} : TON;
   //    TON_3 { ExternalWritable := 'False'} : TON;
   //    TON_4 { ExternalWritable := 'False'} : TON;
   // END_VAR
BEGIN
END_DATA_BLOCK

DATA_BLOCK "n0094-ug7-xn10_SN51_1"   // DB1148, F_DB
VERSION : 0.1
// stored: AutoNumber true, DBAccessibleFromOPCUA true, DBAccessibleFromWebserver true, InstanceOfName 00_Push-Button_Input, InstanceOfType FB
"00_Push-Button_Input"
   // VAR_INPUT
   //    IN_1 : Bool;
   //    IN_2 : Bool;
   //    IN_3 : Bool;
   //    IN_4 : Bool;
   //    ON_Tristate : Bool;
   //    ON_Lamp : Bool;
   //    Reset : Bool;
   //    REAC_DELAY { ExternalWritable := 'False'} : Time;
   //    Bypass_ET200 : Bool;
   // END_VAR
   // VAR_OUTPUT
   //    OUT_1 : Bool;
   //    OUT_2 : Bool;
   //    OUT_3 : Bool;
   //    OUT_4 : Bool;
   //    Diag_1 : Bool;
   //    Diag_2 : Bool;
   //    Diag_3 : Bool;
   //    Diag_4 : Bool;
   //    Lamp_1 : Bool;
   //    Lamp_2 : Bool;
   //    Lamp_3 : Bool;
   //    Lamp_4 : Bool;
   // END_VAR
   // VAR
   //    ESTOP_1 { S7_SetPoint := 'True'} : ESTOP1;
   //    ESTOP_2 { S7_SetPoint := 'True'} : ESTOP1;
   //    ESTOP_3 { S7_SetPoint := 'True'} : ESTOP1;
   //    ESTOP_4 { S7_SetPoint := 'True'} : ESTOP1;
   //    TON_1 { ExternalWritable := 'False'} : TON;
   //    TON_2 { ExternalWritable := 'False'} : TON;
   //    TON_3 { ExternalWritable := 'False'} : TON;
   //    TON_4 { ExternalWritable := 'False'} : TON;
   // END_VAR
BEGIN
END_DATA_BLOCK

DATA_BLOCK "n0094-ug7-xn10_SN51_2"   // DB1149, F_DB
VERSION : 0.1
// stored: AutoNumber true, DBAccessibleFromOPCUA true, DBAccessibleFromWebserver true, InstanceOfName 00_Push-Button_Input, InstanceOfType FB
"00_Push-Button_Input"
   // VAR_INPUT
   //    IN_1 : Bool;
   //    IN_2 : Bool;
   //    IN_3 : Bool;
   //    IN_4 : Bool;
   //    ON_Tristate : Bool;
   //    ON_Lamp : Bool;
   //    Reset : Bool;
   //    REAC_DELAY { ExternalWritable := 'False'} : Time;
   //    Bypass_ET200 : Bool;
   // END_VAR
   // VAR_OUTPUT
   //    OUT_1 : Bool;
   //    OUT_2 : Bool;
   //    OUT_3 : Bool;
   //    OUT_4 : Bool;
   //    Diag_1 : Bool;
   //    Diag_2 : Bool;
   //    Diag_3 : Bool;
   //    Diag_4 : Bool;
   //    Lamp_1 : Bool;
   //    Lamp_2 : Bool;
   //    Lamp_3 : Bool;
   //    Lamp_4 : Bool;
   // END_VAR
   // VAR
   //    ESTOP_1 { S7_SetPoint := 'True'} : ESTOP1;
   //    ESTOP_2 { S7_SetPoint := 'True'} : ESTOP1;
   //    ESTOP_3 { S7_SetPoint := 'True'} : ESTOP1;
   //    ESTOP_4 { S7_SetPoint := 'True'} : ESTOP1;
   //    TON_1 { ExternalWritable := 'False'} : TON;
   //    TON_2 { ExternalWritable := 'False'} : TON;
   //    TON_3 { ExternalWritable := 'False'} : TON;
   //    TON_4 { ExternalWritable := 'False'} : TON;
   // END_VAR
BEGIN
END_DATA_BLOCK
